# B&R Automation Studio project 8238 (part 8)

#### kgGetMachineAdressW3.st - Ermittelt die Maschinenadresse aus Liniennummer und Maschinentyp
```iecst
(********************************************************************
 * COPYRIGHT -- Herbert Kannegiesser GmbH
 ********************************************************************
 * Library: KGstdLib
 * File: kgGetMachineAdressW3.st
 * Author: hunholz
 * Created: February 08, 2012
 ********************************************************************
 * Implementation of library KGstdLib
 ********************************************************************)

(* Ermittelt die Maschinenadresse aus Liniennummer und Maschinentyp *)
FUNCTION kgGetMachineAdressW3

	_diMachineType ACCESS ADR(MachineType);

	kgGetMachineAdressW3 := 0;

	IF MachineType = kgW3SERVER THEN

		kgGetMachineAdressW3 := 202;

	ELSE

		CASE MachineType OF

			kgW3LOADSYSTEM, kgW3EXTRACTOR, kgW3EXTRACTOR2, kgW3CONVEYOR, kgW3SHAKER, kgW3PROCESS:

				IF LineNumber >= 1 AND LineNumber <= 10 THEN

					kgGetMachineAdressW3 := DINT_TO_USINT(_diMachineType) + LineNumber;

				END_IF

			kgW3WASHER, kgW3IFBOX, kgW3DEVICE, kgW3PCSTATION, kgW3BIT:

				IF LineNumber >= 1 AND LineNumber <= 20 THEN

					kgGetMachineAdressW3 := DINT_TO_USINT(_diMachineType) + LineNumber;

				END_IF

			kgW3DRYER, kgW3SINGLEWASHER:

				IF LineNumber >= 1 AND LineNumber <= 30 THEN

					kgGetMachineAdressW3 := DINT_TO_USINT(_diMachineType) + LineNumber;

				END_IF

		END_CASE

	END_IF

END_FUNCTION
```

#### kgCheckDo.st - Prüfe auf Datenobjekt und erzeuge es ggf. neu
```iecst
(********************************************************************
 * COPYRIGHT -- Herbert Kannegiesser GmbH
 ********************************************************************
 * Library: KGstdLib
 * File: kgCheckDo.st
 * Author: hunholz
 * Created: February 22, 2012
 ********************************************************************
 * Implementation of library KGstdLib
 ********************************************************************)

(* Prüfe auf Datenobjekt und erzeuge es ggf. neu *)
FUNCTION_BLOCK kgCheckDo

	IF Enable THEN

		_xReady := FALSE;

		IF MinLen > NomLen THEN

			Status := KG_ERR_WRONGSIZES;
			RETURN;

		END_IF

		REPEAT

			CASE _wStep OF

				0:	// Hole Info

					_doInfo(enable := TRUE, pName := pName);

					IF _doInfo.status = ERR_OK THEN

						IF _doInfo.len >= MinLen THEN

							doId 	:= _doInfo.ident;
							doMem 	:= _doInfo.pDatObjMem;
							doLen 	:= _doInfo.len;

							Status := ERR_OK;

							_xReady := TRUE;

						ELSE

							_wStep := 1;
							Status := ERR_OK;

						END_IF

					ELSIF _doInfo.status <> ERR_FUB_BUSY THEN

						IF Create THEN

							// DO ist nicht vorhanden

							_wStep := 2;
							Status := ERR_OK;

						ELSE

							Status := _doInfo.status;
							_xReady := TRUE;

						END_IF

					END_IF

				1:	// Lösche vorhandenes DO

					_doDelete(enable := TRUE, ident := _doInfo.ident);

					IF _doDelete.status <> ERR_FUB_BUSY THEN

						Status := ERR_OK;
						_wStep := 2;

					ELSE

						Status := ERR_FUB_BUSY;

					END_IF

				2:	// Erzeuge DO neu

					_doCreate(enable := TRUE, grp := 0, pName := pName, len := NomLen, MemType := MemType, Option := 0, pCpyData := 0);

					IF _doCreate.status = ERR_OK THEN

						_wStep := 3;

					ELSIF _doCreate.status <> ERR_FUB_BUSY THEN

						_wStep := 0;

					END_IF

					Status := _doCreate.status;

				3: // Info erneut einlesen

					_doInfo(enable := TRUE, pName := pName);

					IF _doInfo.status = ERR_OK THEN

						doId 	:= _doInfo.ident;
						doMem 	:= _doInfo.pDatObjMem;
						doLen 	:= _doInfo.len;

						Status := KG_INFO_DO_NEW;

						_xReady := TRUE;

						_wStep := 0;

					ELSIF _doInfo.status <> ERR_FUB_BUSY THEN

						Status := _doInfo.status;
						_wStep := 0;

					ELSE

						Status := _doInfo.status;

					END_IF

				ELSE

					_wStep := 0;
					Status := ERR_OK;

			END_CASE

			UNTIL

			Status <> ERR_OK OR _xReady

		END_REPEAT

	ELSE

		_wStep := 0;

		Status := ERR_FUB_ENABLE_FALSE;

	END_IF

END_FUNCTION_BLOCK
```

#### kgXOR.st - XOR über Byte-Feld
```iecst
(********************************************************************
 * COPYRIGHT -- Herbert Kannegiesser GmbH
 ********************************************************************
 * Library: KGstdLib
 * File: kgXOR.st
 * Author: hunholz
 * Created: March 07, 2012
 ********************************************************************
 * Implementation of library KGstdLib
 ********************************************************************)

(* XOR über Byte-Feld *)
FUNCTION kgXOR

	_xStatusOk := pStatus > 0;

	kgXOR := 0;

	IF _xStatusOk THEN
		_wDynStatus ACCESS pStatus;
		_wDynStatus := ERR_OK;
	END_IF

	_xWordResultOk := pWordResult > 0;

	IF _xWordResultOk THEN

		_bWordResult ACCESS pWordResult;

	END_IF

	IF pMem = 0 THEN
		IF _xStatusOk THEN
			_wDynStatus := KG_ERR_NULPOINTER;
		END_IF
		RETURN;

	ELSE

		_bMem ACCESS pMem;

	END_IF

	kgXOR := bInit;

	FOR _i := 1 TO wLen DO

		kgXOR := kgXOR XOR _bMem[_i];

	END_FOR

	IF _xWordResultOk THEN

		_bWordResult[0] := kgXOR;
		_bWordResult[1] := kgXOR;

	END_IF

END_FUNCTION
```

#### kgUnitconfREALtoDisplay.st - Wandelt Wert entsprechend der Unit
```iecst
(********************************************************************
 * COPYRIGHT -- Herbert Kannegiesser GmbH
 ********************************************************************
 * Library: KGstdLib
 * File: kgUnitconfREALtoDisplay.st
 * Author: hunholz
 * Created: March 15, 2012
 ********************************************************************
 * Implementation of library KGstdLib
 ********************************************************************)

(* Wandelt Wert entsprechend der Unit *)
FUNCTION kgUnitconfREALtoDisplay

	lDigits := 0;
	sUnit := '';

	CASE Unit OF

		2,60,70,80,91,901:

			// 1/10
			kgUnitconfREALtoDisplay := Value * 0.1;
			lDigits := 1;

			CASE Unit OF

				2:
					// Sekunden
					sUnit := 's';

				60:
					// Hertz
					sUnit := 'Hz';

				70:
					// Winkel
					sUnit := '°';

				80:
					// Prozent
					sUnit := '%';
				91:
					// Prozent
					sUnit := 'g';

			END_CASE

		90,902:
			// 1/100
			kgUnitconfREALtoDisplay := Value * 0.01;
			lDigits := 2;

			CASE Unit OF

				90:
					// g
					sUnit := 'g';

			END_CASE

		4,903:

			// 1/1000
			kgUnitconfREALtoDisplay := Value * 0.001;
			lDigits := 3;

			CASE Unit OF

				4:
					// Sekunde
					sUnit := 's';

			END_CASE

		10:
			// liter Gallonen
			IF LocUnit = KG_UNIT_US THEN
				kgUnitconfREALtoDisplay := Value * 0.2641721;
				lDigits := 1;
				sUnit := 'US gal';
			ELSE
				kgUnitconfREALtoDisplay := Value;
				sUnit := 'l';
			END_IF

		11:
			// milliliter Ounce
			IF LocUnit = KG_UNIT_US THEN
				kgUnitconfREALtoDisplay := Value * 0.03381402;
				lDigits := 3;
				sUnit := 'fl.Oz.';

			ELSE
				kgUnitconfREALtoDisplay := Value;
				sUnit := 'ml';
			END_IF

		20:
			// mm inch
			IF LocUnit = KG_UNIT_US THEN
				kgUnitconfREALtoDisplay := Value * 0.03937;
				lDigits := 2;
				sUnit := 'inch';
			ELSE
				kgUnitconfREALtoDisplay := Value;
				sUnit := 'mm';
			END_IF

		21:
			// mm cm inch
			IF LocUnit = KG_UNIT_US THEN
				kgUnitconfREALtoDisplay := Value * 0.03937;
				lDigits := 2;
				sUnit := 'inch';
			ELSE
				kgUnitconfREALtoDisplay := Value * 0.1;
				lDigits := 1;
				sUnit := 'cm';
			END_IF

		22:
			// mm dm inch
			IF LocUnit = KG_UNIT_US THEN
				kgUnitconfREALtoDisplay := Value * 0.03937;
				sUnit := 'inch';
			ELSE
				kgUnitconfREALtoDisplay := Value * 0.01;
				sUnit := 'dm';
			END_IF
			lDigits := 2;

		23:
			// mm m feet
			IF LocUnit = KG_UNIT_US THEN
				kgUnitconfREALtoDisplay := Value * 0.00328;
				sUnit := 'ft';
			ELSE
				kgUnitconfREALtoDisplay := Value * 0.001;
				sUnit := 'm';
			END_IF
			lDigits := 3;

		30:
			// 0,1kg kg lbs
			IF LocUnit = KG_UNIT_US THEN
				kgUnitconfREALtoDisplay := Value * 0.220462;
				sUnit := 'lbs';
			ELSE
				kgUnitconfREALtoDisplay := Value * 0.1;
				sUnit := 'kg';
			END_IF
			lDigits := 1;

		40:
			// 0,1 °C °C °F
			IF LocUnit = KG_UNIT_US THEN
				kgUnitconfREALtoDisplay := (Value * 0.18) + 32.0;
				sUnit := '°F';
			ELSE
				kgUnitconfREALtoDisplay := Value * 0.1;
				sUnit := '°C';
			END_IF
			lDigits := 1;

		41:
			// °C °C °F
			IF LocUnit = KG_UNIT_US THEN
				kgUnitconfREALtoDisplay := (Value * 1.8) + 32.0;
				sUnit := '°F';
			ELSE
				kgUnitconfREALtoDisplay := Value;
				sUnit := '°C';
			END_IF

		50:
			// 0,1 bar bar psi
			IF LocUnit = KG_UNIT_US THEN
				kgUnitconfREALtoDisplay := Value * 1.450368;
				sUnit := 'psi';
			ELSE
				kgUnitconfREALtoDisplay := Value * 0.1;
				lDigits := 1;
				sUnit := 'bar';
			END_IF

		310:
			// 0,01 l/kg l/kg gal/lbs
			IF LocUnit = KG_UNIT_US THEN
				kgUnitconfREALtoDisplay := Value * 0.00119827;
				lDigits := 2;
				sUnit := 'gal/lbs';
			ELSE
				kgUnitconfREALtoDisplay := Value * 0.01;
				lDigits := 1;
				sUnit := 'l/kg';
			END_IF

		ELSE

			kgUnitconfREALtoDisplay := Value;

			CASE Unit OF

				1:
					sUnit := 's';
				3:
					sUnit := 'min';
				81:
					sUnit := '%';

			END_CASE

	END_CASE

	IF pDigits > 0 THEN

		brsmemcpy(pDigits, ADR(lDigits), SIZEOF(lDigits));

	END_IF

	IF pUnit > 0 THEN

		brsmemcpy(pUnit, ADR(sUnit), SIZEOF(sUnit));

	END_IF

END_FUNCTION
```

#### kgUnitconfDisplayToREAL.st - Wandelt Wert entsprechend der Unit
```iecst
(********************************************************************
 * COPYRIGHT -- Herbert Kannegiesser GmbH
 ********************************************************************
 * Library: KGstdLib
 * File: kgUnitconfDisplayToREAL.st
 * Author: hunholz
 * Created: March 15, 2012
 ********************************************************************
 * Implementation of library KGstdLib
 ********************************************************************)

(* Wandelt Wert entsprechend der Unit *)
FUNCTION kgUnitconfDisplayToREAL

	CASE Unit OF

		2,60,70,80,91,901:
			// 1/10
			kgUnitconfDisplayToREAL := Display * 10;

		90,902:
			// 1/100
			kgUnitconfDisplayToREAL := Display * 100;

		4,903:
			// 1/1000
			kgUnitconfDisplayToREAL := Display * 1000;

		10:
			// liter Gallonen
			IF LocUnit = KG_UNIT_US THEN
				kgUnitconfDisplayToREAL := Display / 0.2641721;
			ELSE
				kgUnitconfDisplayToREAL := Display;
			END_IF

		11:
			// milliliter Ounce
			IF LocUnit = KG_UNIT_US THEN
				kgUnitconfDisplayToREAL := Display / 0.03381402;
			ELSE
				kgUnitconfDisplayToREAL := Display;
			END_IF

		20:
			// mm inch
			IF LocUnit = KG_UNIT_US THEN
				kgUnitconfDisplayToREAL := Display / 0.03937;
			ELSE
				kgUnitconfDisplayToREAL := Display;
			END_IF

		21:
			// mm cm inch
			IF LocUnit = KG_UNIT_US THEN
				kgUnitconfDisplayToREAL := Display / 0.03937;
			ELSE
				kgUnitconfDisplayToREAL := Display * 10;
			END_IF

		22:
			// mm dm inch
			IF LocUnit = KG_UNIT_US THEN
				kgUnitconfDisplayToREAL := Display / 0.03937;
			ELSE
				kgUnitconfDisplayToREAL := Display * 100;
			END_IF

		23:
			// mm m feet
			IF LocUnit = KG_UNIT_US THEN
				kgUnitconfDisplayToREAL := Display / 0.00328;
			ELSE
				kgUnitconfDisplayToREAL := Display * 1000;
			END_IF

		30:
			// 0,1kg kg lbs
			IF LocUnit = KG_UNIT_US THEN
				kgUnitconfDisplayToREAL := Display / 0.220462;
			ELSE
				kgUnitconfDisplayToREAL := Display * 10;
			END_IF

		40:
			// 0,1 °C °C °F
			IF LocUnit = KG_UNIT_US THEN
				kgUnitconfDisplayToREAL := (Display - 32.0) / 0.18;
			ELSE
				kgUnitconfDisplayToREAL := Display * 10;
			END_IF

		41:
			// °C °C °F
			IF LocUnit = KG_UNIT_US THEN
				kgUnitconfDisplayToREAL := (Display - 32.0) / 1.8;
			ELSE
				kgUnitconfDisplayToREAL := Display;
			END_IF

		50:
			// 0,1 bar bar psi
			IF LocUnit = KG_UNIT_US THEN
				kgUnitconfDisplayToREAL := Display / 1.450368;
			ELSE
				kgUnitconfDisplayToREAL := Display * 10;
			END_IF

		310:
			// 0,01 l/kg l/kg gal/lbs
			IF LocUnit = KG_UNIT_US THEN
				kgUnitconfDisplayToREAL := Display / 0.00119827;
			ELSE
				kgUnitconfDisplayToREAL := Display * 100;
			END_IF

		ELSE

			kgUnitconfDisplayToREAL := Display;

	END_CASE

END_FUNCTION
```

#### kgGetProgdata.st - Read Programdata from a dataobject
```iecst
(********************************************************************
 * COPYRIGHT -- Herbert Kannegiesser GmbH
 ********************************************************************
 * Library: KGstdLib
 * File: kgGetProgdata.st
 * Author: hunholz
 * Created: April 11, 2012
 ********************************************************************
 * Implementation of library KGstdLib
 ********************************************************************)

(* Read Programdata from a dataobject *)
FUNCTION kgGetProgdata

	IF LEN(sBaseName) = 0 THEN
		kgGetProgdata := KG_ERR_NULLSTRING;
		RETURN;
	END_IF

	IF pMem = 0 THEN
		kgGetProgdata := KG_ERR_NULPOINTER;
		RETURN;
	END_IF

	_sIndex := '';
	IF wProgMaxNo > 9999 AND  wProgNo  < 10000 THEN
		_sIndex := CONCAT(_sIndex,'0');
	END_IF
	IF wProgMaxNo > 999 AND  wProgNo  < 1000 THEN
		_sIndex := CONCAT(_sIndex,'0');
	END_IF
	IF wProgMaxNo > 99 AND  wProgNo  < 100 THEN
		_sIndex := CONCAT(_sIndex,'0');
	END_IF
	IF wProgMaxNo > 9 AND  wProgNo  < 10 THEN
		_sIndex := CONCAT(_sIndex,'0');
	END_IF

	_sIndex1 := UINT_TO_STRING(wProgNo);

	_sIndex := CONCAT(_sIndex, _sIndex1);

	_sName := CONCAT(sBaseName, _sIndex);

	_diProg(enable := TRUE, pName := ADR(_sName));

	IF _diProg.status = ERR_OK THEN

		// Bug 690 : Datenobjekt hat 4Byte Alignment. Struktur kann 1 bis 3 Byte kleiner sein.
//		IF _diProg.len > lSize THEN
//			kgGetProgdata := KG_ERR_WRONGSIZES;
//			RETURN;
//		END_IF

		brsmemcpy(pMem, _diProg.pDatObjMem, MIN(_diProg.len,lSize));

		kgGetProgdata := ERR_OK;

		RETURN;

	ELSE
		kgGetProgdata := _diProg.status;
		RETURN;
	END_IF

END_FUNCTION
```

#### kgSignalLight.st - Process red/yellow/green
```iecst
(********************************************************************
 * COPYRIGHT -- Herbert Kannegiesser GmbH
 ********************************************************************
 * Library: KGstdLib
 * File: kgSignalLight.st
 * Author: hunholz
 * Created: July 12, 2012
 ********************************************************************
 * Implementation of library KGstdLib
 ********************************************************************)

(* Process red/yellow/green *)
FUNCTION kgSignalLight

	xGreen 		:= FALSE;
	xRed		:= FALSE;
	xYellow 	:= FALSE;

	CASE wStatus OF

		(*-0- Maschine aus*)
		KG_MACHINESTATE_OFF:

		(*-1- NOT-HALT*)
		KG_MACHINESTATE_EMERGENCYSTOP:

			xRed := xClock;

		(*-2- Sicherer HALT*)
		KG_MACHINESTATE_SAFESTOP:

			xYellow := xClock;

		(*-3- Störung*)
		KG_MACHINESTATE_FAULT:

			xRed := TRUE;

		(*-4- Störung quittierbar*)
		KG_MACHINESTATE_FAULT_GONE:

			xRed := TRUE;
			xYellow := xClock;

		(*-5- Service / Handbetrieb*)
		KG_MACHINESTATE_SERVICE:

			xYellow := xClock;
			xGreen := xClock;

		(*-6- Maschine läuft*)
		KG_MACHINESTATE_AUTOMATIC_RUN:

			xGreen := TRUE;

		(*-7- STOP*)
		KG_MACHINESTATE_STOP:

		(*-8- Maschine wartet auf Automatik-Freigabe*)
		KG_MACHINESTATE_WAIT_AUTOMATIC:

			xGreen := xClock;

		(*-9- Maschine wartet auf Bestätigung durch Bediener*)
		KG_MACHINESTATE_WAIT_MAN:

			xYellow := xClock;
			xGreen := TRUE;

		(*-10- Warnung*)
		KG_MACHINESTATE_WARNING:

			xYellow := TRUE;
			xGreen := TRUE;

		ELSE

			xGreen := TRUE;

	END_CASE

END_FUNCTION
```

### KGStandard-History.txt
```
1.00.0	30.06.2011 NEU
1.01.0	02.07.2011 mnCnt ergänzt
1.02.0	08.07.2011 Netlink 1.02.0
1.03.0  19.07.2011 kgStd 1.01.0
1.04.0	26.07.2011 Maschinentyp in der Infostruktur auf 11 Zeichen verringert
1.05.0		   Keine Ahnung
1.06.0	01.09.2011 Info_typ erweitert
1.07.0	20.09.2011 Stat_typ ergänzt
1.08.0	06.10.2011 Netlink 1.05.0
1.08.1	14.10.2011 Netlink 1.06.0
1.09.0  03.11.2011 Umstellung auf AS 3.0.90
					- Stat_typ erweitert
					- Funktionen zum Generieren einer Postennummer in KGstdLib ergänzt 1.02.0
1.10.0	20.12.2011 Ringbufferfunktionen ergänzt
				   KGBOM ergänzt
				   KG_DEVICE_COMPACTFLASH ergänzt
1.11.0	03.01.2012 kgGUIDisZero : Funktion prüft, ob eine GUID null ist.
1.12.0	12.01.2012 kgNextBatchNoLong merkt sich die letzte Postennummer. BatchNo ist nur noch Output.
1.13.0	24.01.2012 Erweiterung der Ringbuffer-Funktionen. Einführung des Startzeigers.
				   Unabhängigkeit von Netlink. Netlink entfernt.
				   Konstanten für Maschinenstati ergänzt
				   Maschinentypen aus NetLink-Library übernommen. nlMachinetypeW3_typ --> kgMachinetypeW3_typ
				   Datentypen utfName15 und utfName31 als abgeleiteten Datentyp deklariert
1.14.0	03.02.2012 Im Pkg_KGStandardShare werden die Konstanten KG_DEVICE_USBSTICK1 und KG_DEVICE_USBSTICK2 als STRING[31] deklariert.
				   In der sysconf sollten die Device-Namen für gültige USB-Massenspeicher definiert sein.
1.15.0	08.02.2012 Funktionen: kgGetLineNumberW3 und kgGetMachineAdressW3. (mnEth Version 2.08.0 verwenden)
1.15.1	15.02.2012 kgGetBatchNoUnique und kgNextBatchNoLong korrigiert
1.16.0	15.03.2012 Konvertierung von Parametern entsprechend der Einheit (units.csv 2011-11-25T08:56:00)
1.16.1	15.03.2012 Für Displaywerte werden auch die Nachkommastellen mit angegeben
1.16.2	20.03.2012 Bugfix KGstdLib
1.17.0	21.03.2012 KGstdLib erweitert
1.17.1	22.03.2012 CP3585 ergänzt
1.18.0	04.04.2012 _Info_ gibt es nicht mehr
1.19.0	11.04.2012 Enumeration für Maschinenstati
1.20.0	04.05.2012 Einheit (91) 0,1 g ergänzt
1.21.0	18.06.2012 CP1584 ergänzt
		19.06.2012 Bug 690: Programm lässt sich nicht laden behoben
		21.06.2012 Maschinenstati in Hex-Notation und als USINT. Erweiterter Maschinenstatus als UINT mit Bit 8 für Stop und Bit 9 für Warten
1.22.0	25.06.2012 Module Identifier ergänzt (X20DI9371, X20DO9322)
1.23.0	03.07.2012 Module Identifier ergänzt (X20IF1072, X20IF2772, X20BR9300, X20PS2100, 4PP065IF231
1.24.0	18.07.2012 Module Identifier ergänzt (X20BT9400, X67DM1321
1.25.0	18.09.2012 CP3484 ergänzt
```

### Package Logical/Standard/Kanlink/KGFramework/Pkg_mnSystem - Systemtask für Versionierung

### Program Logical/Standard/Kanlink/KGFramework/Pkg_mnSystem/mnSystem (IEC) - Systemtask für Versionierung

#### mnSystemCyclic.st - Cyclic code
```iecst
(********************************************************************
 * COPYRIGHT -- Kannegiesser GmbH
 ********************************************************************
 * Program: mnSystem
 * File: mnSystemCyclic.st
 * Author: Hunholz
 * Created: Mar 16, 2012
 ********************************************************************
 * Implementation of program mnSystem
 ********************************************************************)

PROGRAM _CYCLIC

	//**********************
	// USB Knoten überwachen
	//**********************

	// Alle 5 Sekunden eine Liste der verfügbaren Sticks zur Verfügung stellen

	_TONsearchForUSB(IN := _wUSBstate = 0 , PT := T#5s);

	CASE _wUSBstate OF

		0:

			IFmnSystem.Out.sInterfaceUSB := _sInterfaceUSB;
			IFmnSystem.Out.xUSBStickReady := _xUSBStickReady;

			IF _TONsearchForUSB.Q OR _xFirstScan THEN

				_xFirstScan := FALSE;
				_wUSBstate := 1;

			END_IF

		1:
			_UsbNodeListGet(enable := TRUE, pBuffer := ADR(_lUSBlist), bufferSize := SIZEOF(_lUSBlist), filterInterfaceClass := asusb_CLASS_MASS_STORAGE, filterInterfaceSubClass := asusb_SUBCLASS_SCSI_COMMAND_SET);

			IF _UsbNodeListGet.status <> ERR_FUB_BUSY THEN

				_sInterfaceUSB := '';
				_xUSBStickReady := FALSE;

				IF _UsbNodeListGet.status = ERR_OK THEN

					_wUSBstate := 2;

					_wCycleFound := _wCycleFound + 1;

				ELSE

					IFmnSystem.Out.xUSBStickScanned := TRUE;
					_wUSBstate := 0;

					_wCycleNotFound := _wCycleNotFound + 1;

				END_IF

			END_IF

		2:

			_UsbNodeGet(enable := TRUE, nodeId := _lUSBlist[1], pBuffer := ADR(_usbNode), bufferSize := SIZEOF(_usbNode));

			IF _UsbNodeGet.status <> ERR_FUB_BUSY THEN

				IF _UsbNodeGet.status = ERR_OK THEN

					brsmemcpy(ADR(_sInterfaceUSB),ADR(_usbNode.ifName),SIZEOF(_sInterfaceUSB));
					_xUSBStickReady := TRUE;

					_wCycleReady := _wCycleReady + 1;

				END_IF

				IFmnSystem.Out.xUSBStickScanned := TRUE;
				IFmnSystem.Out.sInterfaceUSB := _sInterfaceUSB;
				IFmnSystem.Out.xUSBStickReady := _xUSBStickReady;

				_wUSBstate := 0;

			END_IF

		ELSE

			_wUSBstate := 0;

	END_CASE

	//#####################################################################################################################

	// Heartbeeat erzeugen (Sekunden)
	_GetTime(enable := TRUE);
	mnSystemStatAd.wHeartbeat := DT_TO_UINT(_GetTime.DT1);

	_diDifSystime := IFmnSystem.In.PLC.diSystemTime - _diOldSysTime;
	_diOldSysTime := IFmnSystem.In.PLC.diSystemTime;

	IF _diDifSystime >= 0 THEN

		_l1sCount := _l1sCount + DINT_TO_UDINT(_diDifSystime);

		IF _l1sCount > 1000000 THEN

			IFmnSystem.Out.x1s := NOT IFmnSystem.Out.x1s;
			_l1sCount := _l1sCount - 1000000;

		END_IF

		_l500msCount := _l500msCount + DINT_TO_UDINT(_diDifSystime);

		IF _l500msCount > 500000 THEN

			IFmnSystem.Out.x500ms := NOT IFmnSystem.Out.x500ms;
			_l500msCount := _l500msCount - 500000;

		END_IF

	END_IF

	// Lüfterüberwachung

	CASE IFmnSystem.In.PLC.wMDL_ID OF

		KG_CPU_X20CP1486:

			_xFanOk := IFmnSystem.In.PLC.xFanOk;

		ELSE

			_xFanOk := TRUE;

	END_CASE

	//********************************
	// Überwachung Umgebungstemperatur
	//********************************

	_TONtemp(IN := (IFmnSystem.In.PLC.wTemperatureENV > mnSystemPar.Mac.wWarnTemperatureEnvironment) AND IFmnParam.Out.xParamOK, PT := T#10m);
	_TONtempC(IN := (IFmnSystem.In.PLC.wTemperatureENV > (mnSystemPar.Mac.wWarnTemperatureEnvironment - 50)) AND IFmnParam.Out.xParamOK, PT := T#10m);

	//************************
	// Überwachung von Modulen
	//************************

	IF IFmnParam.Out.xParamOK THEN

		_xModuleFault := FALSE;
		_wModuleFaultLineNumber := 0;
		_wModuleFaultModuleNumber := 0;

		FOR _ii := 1 TO MNSYSTEM_CNT_MODULELINES DO

			FOR _jj := 1 TO MNSYSTEM_CNT_MODULES DO

				IF mnSystemPar.Cfg.Lines[_ii].wModuleID[_jj] <> KG_MODULE_NO THEN

					// Modul ist konfiguriert

					IF (mnSystemPar.Cfg.Lines[_ii].wModuleID[_jj] <> IFmnSystem.In.ModuleInfo[_ii,_jj].wMDL_ID) THEN
						_xModuleFault := TRUE;
						_wModuleFaultLineNumber := _ii;
						_wModuleFaultModuleNumber := _jj;
						EXIT;
					END_IF

				END_IF

			END_FOR

			IF _xModuleFault THEN
				EXIT;
			END_IF

		END_FOR

		// Cooling

		FOR _iC := 1 TO 2 DO

			IF NOT _xCInitDone[_iC] THEN

				IF mnSystemPar.Cfg.BindingMotProtCooling[_iC].wBindIndexModul > 0 AND mnSystemPar.Cfg.BindingMotProtCooling[_iC].wBindIndexModul <= MNSYSTEM_CNT_MODULES
					AND mnSystemPar.Cfg.BindingMotProtCooling[_iC].wBindIndexChannel > 0 AND mnSystemPar.Cfg.BindingMotProtCooling[_iC].wBindIndexChannel <= 12 THEN

					_BindMotProtCooling[_iC].wModule := mnSystemPar.Cfg.BindingMotProtCooling[_iC].wBindIndexModul;
					_BindMotProtCooling[_iC].wChannel := mnSystemPar.Cfg.BindingMotProtCooling[_iC].wBindIndexChannel;
					_BindMotProtCooling[_iC].sDiscription := mnSystemPar.Cfg.BindingMotProtCooling[_iC].sDiscription;
					_BindMotProtCooling[_iC].xInvers := mnSystemPar.Cfg.BindingMotProtCooling[_iC].xInvers;
					_BindMotProtCooling[_iC].xQualitiyOk := TRUE;

				END_IF

				IF mnSystemPar.Cfg.BindingOutCooling[_iC].wBindIndexModul > 0 AND mnSystemPar.Cfg.BindingOutCooling[_iC].wBindIndexModul <= MNSYSTEM_CNT_MODULES
					AND mnSystemPar.Cfg.BindingOutCooling[_iC].wBindIndexChannel > 0 AND mnSystemPar.Cfg.BindingOutCooling[_iC].wBindIndexChannel <= 12 THEN

					_BindingOutCooling[_iC].wModule := mnSystemPar.Cfg.BindingOutCooling[_iC].wBindIndexModul;
					_BindingOutCooling[_iC].wChannel := mnSystemPar.Cfg.BindingOutCooling[_iC].wBindIndexChannel;
					_BindingOutCooling[_iC].sDiscription := mnSystemPar.Cfg.BindingOutCooling[_iC].sDiscription;
					_BindingOutCooling[_iC].xInvers := mnSystemPar.Cfg.BindingOutCooling[_iC].xInvers;
					_BindingOutCooling[_iC].xQualitiyOk := TRUE;

				END_IF

				IF mnSystemPar.Cfg.BindingWarnEnvTemp[_iC].wBindIndexModul > 0 AND mnSystemPar.Cfg.BindingWarnEnvTemp[_iC].wBindIndexModul <= MNSYSTEM_CNT_MODULES
					AND mnSystemPar.Cfg.BindingWarnEnvTemp[_iC].wBindIndexChannel > 0 AND mnSystemPar.Cfg.BindingWarnEnvTemp[_iC].wBindIndexChannel <= 12 THEN

					_BindingWarnEnvTemp[_iC].wModule := mnSystemPar.Cfg.BindingWarnEnvTemp[_iC].wBindIndexModul;
					_BindingWarnEnvTemp[_iC].wChannel := mnSystemPar.Cfg.BindingWarnEnvTemp[_iC].wBindIndexChannel;
					_BindingWarnEnvTemp[_iC].sDiscription := mnSystemPar.Cfg.BindingWarnEnvTemp[_iC].sDiscription;
					_BindingWarnEnvTemp[_iC].xInvers := mnSystemPar.Cfg.BindingWarnEnvTemp[_iC].xInvers;
					_BindingWarnEnvTemp[_iC].xQualitiyOk := TRUE;

				END_IF

				_xCInitDone[_iC] := TRUE;

			ELSE

				IF _BindMotProtCooling[_iC].xQualitiyOk THEN

					_xFaultMotProtCooling[_iC] := MDLIn[1,_BindMotProtCooling[_iC].wModule].xIn[_BindMotProtCooling[_iC].wChannel] XOR _BindMotProtCooling[_iC].xInvers;

				ELSE

					_xFaultMotProtCooling[_iC] := FALSE;

				END_IF

				IF _BindingWarnEnvTemp[_iC].xQualitiyOk THEN

					_xWarnEnvTemp[_iC] := MDLIn[1,_BindingWarnEnvTemp[_iC].wModule].xIn[_BindingWarnEnvTemp[_iC].wChannel] XOR _BindingWarnEnvTemp[_iC].xInvers;

				ELSE

					_xWarnEnvTemp[_iC] := FALSE;

				END_IF

				IF _BindingOutCooling[_iC].xQualitiyOk THEN

					MDLOut[1,_BindingOutCooling[_iC].wModule].xOut[_BindingOutCooling[_iC].wChannel] := (NOT _xFaultMotProtCooling[_iC] AND (_xWarnEnvTemp[_iC] OR (_TONtempC.Q AND (_iC = 1))))
																											XOR _BindingOutCooling[_iC].xInvers;

				END_IF

			END_IF

		END_FOR

	ELSE

		_xModuleFault := FALSE;
		_wModuleFaultLineNumber := 0;
		_wModuleFaultModuleNumber := 0;

	END_IF

	// Meldungen
	IF NOT IFmnTest.Out.xNoMessages THEN

		kgMsgStatus[MNSYSTEM_IDX_KGMSGSTAT].wFunction_ID 	:= 110;

		IF _xModuleFault THEN

			kgMsgStatus[MNSYSTEM_IDX_KGMSGSTAT].wMsgClass		:= MNMSG_CLASS_WARNING;
			kgMsgStatus[MNSYSTEM_IDX_KGMSGSTAT].wMsgAckLevel	:= 0;
			kgMsgStatus[MNSYSTEM_IDX_KGMSGSTAT].wMsgNumber		:= MNSYSTEM_MSG_WRONGMODULE;
			kgMsgStatus[MNSYSTEM_IDX_KGMSGSTAT].diMsgAttr1		:= _wModuleFaultLineNumber;
			kgMsgStatus[MNSYSTEM_IDX_KGMSGSTAT].diMsgAttr2		:= _wModuleFaultModuleNumber;
			kgMsgStatus[MNSYSTEM_IDX_KGMSGSTAT].sMsgAttrTxt		:= mnSystemPar.Cfg.Lines[_wModuleFaultLineNumber].sName[_wModuleFaultModuleNumber];

		ELSIF NOT _xFanOk THEN

			kgMsgStatus[MNSYSTEM_IDX_KGMSGSTAT].wMsgClass		:= MNMSG_CLASS_WARNING;
			kgMsgStatus[MNSYSTEM_IDX_KGMSGSTAT].wMsgAckLevel	:= 0;
			kgMsgStatus[MNSYSTEM_IDX_KGMSGSTAT].wMsgNumber		:= MNSYSTEM_MSG_FAN;
			kgMsgStatus[MNSYSTEM_IDX_KGMSGSTAT].diMsgAttr1		:= 0;
			kgMsgStatus[MNSYSTEM_IDX_KGMSGSTAT].diMsgAttr2		:= 0;
			kgMsgStatus[MNSYSTEM_IDX_KGMSGSTAT].sMsgAttrTxt		:= '';

		ELSIF _xFaultMotProtCooling[1] OR _xFaultMotProtCooling[1] THEN

			kgMsgStatus[MNSYSTEM_IDX_KGMSGSTAT].wMsgClass		:= MNMSG_CLASS_WARNING;
			kgMsgStatus[MNSYSTEM_IDX_KGMSGSTAT].wMsgAckLevel	:= 0;
			kgMsgStatus[MNSYSTEM_IDX_KGMSGSTAT].wMsgNumber		:= MNSYSTEM_MSG_MOTPROTCOOLING;
			kgMsgStatus[MNSYSTEM_IDX_KGMSGSTAT].diMsgAttr1		:= 0;
			kgMsgStatus[MNSYSTEM_IDX_KGMSGSTAT].diMsgAttr2		:= 0;
			IF _xFaultMotProtCooling[1] THEN
				kgMsgStatus[MNSYSTEM_IDX_KGMSGSTAT].sMsgAttrTxt		:= _BindMotProtCooling[1].sDiscription;
			ELSE
				kgMsgStatus[MNSYSTEM_IDX_KGMSGSTAT].sMsgAttrTxt		:= _BindMotProtCooling[2].sDiscription;
			END_IF

		ELSIF _TONtemp.Q OR _xWarnEnvTemp[1] OR _xWarnEnvTemp[2] THEN

			kgMsgStatus[MNSYSTEM_IDX_KGMSGSTAT].wMsgClass		:= MNMSG_CLASS_WARNING;
			kgMsgStatus[MNSYSTEM_IDX_KGMSGSTAT].wMsgAckLevel	:= 0;
			kgMsgStatus[MNSYSTEM_IDX_KGMSGSTAT].wMsgNumber		:= MNSYSTEM_MSG_ENVTEMP;
			kgMsgStatus[MNSYSTEM_IDX_KGMSGSTAT].diMsgAttr1		:= 0;
			kgMsgStatus[MNSYSTEM_IDX_KGMSGSTAT].diMsgAttr2		:= 0;
			IF _xWarnEnvTemp[1] THEN
				kgMsgStatus[MNSYSTEM_IDX_KGMSGSTAT].sMsgAttrTxt		:= mnSystemPar.Cfg.sSwitchBoxName[1];
			ELSIF _xWarnEnvTemp[2] THEN
				kgMsgStatus[MNSYSTEM_IDX_KGMSGSTAT].sMsgAttrTxt		:= mnSystemPar.Cfg.sSwitchBoxName[2];
			ELSE
				kgMsgStatus[MNSYSTEM_IDX_KGMSGSTAT].sMsgAttrTxt		:= 'CPU';
			END_IF

		ELSIF IFmnSystem.In.PLC.bBatteryStatusCPU <> 1 THEN

			kgMsgStatus[MNSYSTEM_IDX_KGMSGSTAT].wMsgClass		:= MNMSG_CLASS_WARNING;
			kgMsgStatus[MNSYSTEM_IDX_KGMSGSTAT].wMsgAckLevel	:= 0;
			kgMsgStatus[MNSYSTEM_IDX_KGMSGSTAT].wMsgNumber		:= MNSYSTEM_MSG_BATTERY;
			kgMsgStatus[MNSYSTEM_IDX_KGMSGSTAT].diMsgAttr1		:= 0;
			kgMsgStatus[MNSYSTEM_IDX_KGMSGSTAT].diMsgAttr2		:= 0;
			kgMsgStatus[MNSYSTEM_IDX_KGMSGSTAT].sMsgAttrTxt		:= '';

		ELSE

			kgMsgStatus[MNSYSTEM_IDX_KGMSGSTAT].wFunction_ID 	:= 110;
			kgMsgStatus[MNSYSTEM_IDX_KGMSGSTAT].wMsgClass		:= 0;
			kgMsgStatus[MNSYSTEM_IDX_KGMSGSTAT].wMsgAckLevel	:= 0;
			kgMsgStatus[MNSYSTEM_IDX_KGMSGSTAT].wMsgNumber		:= 0;
			kgMsgStatus[MNSYSTEM_IDX_KGMSGSTAT].diMsgAttr1		:= 0;
			kgMsgStatus[MNSYSTEM_IDX_KGMSGSTAT].diMsgAttr2		:= 0;
			kgMsgStatus[MNSYSTEM_IDX_KGMSGSTAT].sMsgAttrTxt		:= '';

		END_IF

	END_IF

	// Stati
	mnSystemStatAd.lSerialNumber 			:= IFmnSystem.In.PLC.lSerialNumber;
	mnSystemStatAd.wTemperatureCPU 			:= IFmnSystem.In.PLC.wTemperatureCPU;
	mnSystemStatAd.wTemperatureEnvironment 	:= IFmnSystem.In.PLC.wTemperatureENV;

	// Interface
	IFmnSystem.Out.xModuleFault				:= _xModuleFault;

END_PROGRAM
```

#### mnSystemInit.st - Initialization code
```iecst
(********************************************************************
 * COPYRIGHT -- Kannegiesser GmbH
 ********************************************************************
 * Program: mnSystem
 * File: mnSystemInit.st
 * Author: horn
 * Created: January 10, 2012
 ********************************************************************
 * Implementation of program mnSystem
 ********************************************************************)

PROGRAM _INIT

	// Packet-Version auslesen mit MO_ver aus SYS_lib und für den Additional Status zur Verfügung stellen

	_sPkgName := 'mnSystem';

	IF ( MO_ver(ADR(_sPkgName), 0, ADR(_VerStruc)) = 0 ) THEN

		brsmemcpy(ADR(mnSystemStatAd.sPkgVersion), ADR(_VerStruc.version), SIZEOF(_VerStruc.version));

	ELSE

		mnSystemStatAd.sPkgVersion := '---';

	END_IF

	_sPkgName := 'mnMaster';

	IF ( MO_ver(ADR(_sPkgName), 0, ADR(_VerStruc)) = 0 ) THEN

		brsmemcpy(ADR(mnSystemStatAd.sPrjVersion), ADR(_VerStruc.version), SIZEOF(_VerStruc.version));

	ELSE

		mnSystemStatAd.sPrjVersion := '---';

	END_IF

	_sPkgName := 'mnTest';

	IF ( MO_ver(ADR(_sPkgName), 0, ADR(_VerStruc)) = 0 ) THEN

		brsmemcpy(ADR(mnSystemStatAd.sFWVersion), ADR(_VerStruc.version), SIZEOF(_VerStruc.version));

	ELSE

		mnSystemStatAd.sFWVersion := '---';

	END_IF

	// CPU-Typ bestimmen

	CASE IFmnSystem.In.PLC.wMDL_ID OF

		KG_CPU_CTT_11:

			mnSystemStatAd.sCPUType := 'CTT-11';

		KG_CPU_PCT_03:

			mnSystemStatAd.sCPUType := 'PCT-03';

		KG_CPU_PCT_04:

			mnSystemStatAd.sCPUType := 'PCT-04';

		KG_CPU_PP65_0571_P74:

			mnSystemStatAd.sCPUType := 'PP65.0571.P74';

		KG_CPU_PP420_1043_75:

			mnSystemStatAd.sCPUType := 'PP420.1043.75';

		KG_CPU_X20CP1484:

			mnSystemStatAd.sCPUType := 'CP1484';

		KG_CPU_X20CP1484_1:

			mnSystemStatAd.sCPUType := 'CP1484-1';

		KG_CPU_X20CP1486:

			mnSystemStatAd.sCPUType := 'CP1486';

		KG_CPU_X20CP3484:

			mnSystemStatAd.sCPUType := 'CP3484';

		KG_CPU_X20CP3484_1:

			mnSystemStatAd.sCPUType := 'CP3484-1';

		KG_CPU_X20CP3486:

			mnSystemStatAd.sCPUType := 'CP3486';

		KG_CPU_X20CP3585:

			mnSystemStatAd.sCPUType := 'CP3585';

		KG_CPU_X20CP1584:

			mnSystemStatAd.sCPUType := 'CP1584';

		ELSE

			mnSystemStatAd.sCPUType := UINT_TO_STRING(IFmnSystem.In.PLC.wMDL_ID);

	END_CASE

	_wMdlId := IFmnSystem.In.PLC.wMDL_ID;

END_PROGRAM
```

#### mnSystem.typ - Local data types
```iecst
(********************************************************************
 * COPYRIGHT -- Kannegiesser GmbH
 ********************************************************************
 * Program: mnSystem
 * File: _mnSystem.typ
 * Author: horn
 * Created: January 10, 2012
 ********************************************************************
 * Local data types of program mnSystem
 ********************************************************************)

TYPE
	_mnSystemMdlBind_typ : 	STRUCT
		wModule : UINT;
		wChannel : UINT;
		sDiscription : STRING[13];
		xInvers : BOOL;
		xQualitiyOk : BOOL;
	END_STRUCT;
END_TYPE
```

#### mnSystem.var - Local variables
```iecst
(********************************************************************
 * COPYRIGHT -- Kannegiesser GmbH
 ********************************************************************
 * Program: mnSystem
 * File: _mnSystem.var
 * Author: horn
 * Created: January 10, 2012
 ********************************************************************
 * Local variables of program mnSystem
 ********************************************************************)
VAR
	_sPkgName : STRING[11];
	_VerStruc : MoVerStruc_typ;
	_GetTime : DTGetTime;
	_xFanOk : BOOL;
	_wMdlId : UINT;
	_TONtemp : TON;
	_wUSBstate : UINT;
	_TONsearchForUSB : TON;
	_lUSBlist : ARRAY[1..3] OF UDINT;
	_UsbNodeListGet : UsbNodeListGet;
	_sInterfaceUSB : STRING[31];
	_xUSBStickReady : BOOL;
	_usbNode : usbNode_typ;
	_UsbNodeGet : UsbNodeGet;
	_xFirstScan : BOOL := TRUE;
	_wCycleFound : UINT;
	_wCycleNotFound : UINT;
	_wCycleReady : UINT;
	_xModuleFault : BOOL;
	_wModuleFaultLineNumber : UINT;
	_wModuleFaultModuleNumber : UINT;
	_ii : UINT;
	_jj : UINT;
	_iC : UINT;
	_xCInitDone : ARRAY[1..2] OF BOOL;
	_BindMotProtCooling : ARRAY[1..2] OF _mnSystemMdlBind_typ;
	_BindingOutCooling : ARRAY[1..2] OF _mnSystemMdlBind_typ;
	_BindingWarnEnvTemp : ARRAY[1..2] OF _mnSystemMdlBind_typ;
	_xFaultMotProtCooling : ARRAY[1..2] OF BOOL;
	_xWarnEnvTemp : ARRAY[1..2] OF BOOL;
	_TONtempC : TON;
	_diDifSystime : DINT;
	_diOldSysTime : DINT;
	_l1sCount : UDINT;
	_l500msCount : UDINT;
END_VAR
```

### Pkg_mnSystem.typ - Local data types
```iecst
(********************************************************************
 * COPYRIGHT -- Kannegiesser GmbH
 ********************************************************************
 * Program: mnSystem
 * File: mnSystem.typ
 * Author: horn
 * Created: January 10, 2012
 ********************************************************************
 * Local data types of program mnSystem
 ********************************************************************)

TYPE
	mnSystemStatAd_typ : 	STRUCT
		sPkgVersion : STRING[10]; (*Version des Packes mnSystem*)
		sPrjVersion : STRING[10]; (*Hauptversion des Projektes*)
		sFWVersion : STRING[10]; (*Frameworkversion abgeleitet aus mnTest*)
		sCPUType : STRING[19]; (*CPU-Typ*)
		wHeartbeat : UINT; (*Zählt sekündlich hoch*)
		wTemperatureCPU : UINT; (*CPU Temperatur 1/10 °C*)
		wTemperatureEnvironment : UINT; (*Umgebungstemperatur 1/10 °C*)
		lSerialNumber : UDINT; (*Seriennummer der CPU*)
	END_STRUCT;
	IFmnSystem_typ : 	STRUCT
		In : IFmnSystemIn_typ;
		Out : IFmnSystemOut_typ;
	END_STRUCT;
	IFmnSystemOut_typ : 	STRUCT
		xUSBStickReady : BOOL; (*USB-Stick erkannt*)
		xUSBStickScanned : BOOL; (*USB-Stick-Scan wurde erstmals durchgeführt*)
		xModuleFault : BOOL;
		sInterfaceUSB : STRING[31]; (*Interfacebezeichnung für den Stick*)
		x1s : BOOL;
		x500ms : BOOL;
	END_STRUCT;
	IFmnSystemIn_typ : 	STRUCT
		PLC : mnSystem_PLC_typ;
		ModuleInfo : ARRAY[1..MNSYSTEM_CNT_MODULELINES,1..MNSYSTEM_CNT_MODULES]OF mnSystem_ModuleInfo_typ;
		ModuleStatus : ARRAY[1..MNSYSTEM_CNT_MODULELINES,1..MNSYSTEM_CNT_MODULES]OF mnSystem_ModuleStatus_typ;
		xSupplyFault : ARRAY[1..12]OF BOOL;
	END_STRUCT;
	mnSystem_PLC_typ : 	STRUCT
		lSerialNumber : UDINT; (*Serien-Nummer des X20 Moduls*)
		wMDL_ID : UINT; (*Modul-ID des X20 Moduls*)
		bModeSwitch : USINT; (*Version der Firmware*)
		bBatteryStatusCPU : USINT; (*Status der Pufferbatterie*)
		xFanOk : BOOL; (*Status des CPU-Lüfters*)
		wTemperatureCPU : UINT; (*CPU-Temperatur*)
		wTemperatureENV : UINT;
		diSystemTime : DINT; (*Systemzeit der CPU in µs*)
		xStatusInput01 : BOOL; (*Status der 24V-Versorgung für I/O*)
		lPowerOnCycles : UDINT;
		lOperatingHoursPP : UDINT;
	END_STRUCT;
	mnSystem_ModuleStatus_typ : 	STRUCT
		xiMDL_OK : BOOL; (*Status des Moduls*)
		xiStatIn01 : BOOL; (*Busversorgungswarnung (1 = Ueberstrom >2,3 A oder Unterspannung <4,7 V) *)
		xiStatIn02 : BOOL; (*I/O Versorgungswarnung (0 = DC OK)*)
		aiStatus : USINT; (*Status bei Temperatur Modul*)
		xiSingleStatus : ARRAY[1..12]OF BOOL; (*Status bei digitalen Ausgängen*)
	END_STRUCT;
	mnSystem_ModuleInfo_typ : 	STRUCT
		lSerialNumber : UDINT; (*Serien-Nummer des X20 Moduls*)
		wMDL_ID : UINT; (*Modul-ID des X20 Moduls*)
		wHwVariant : UINT; (*Hardware Variante des X20 Moduls*)
		wFirmwareVers : UINT; (*Version der Firmware*)
	END_STRUCT;
	mnSystem_SignalIn_typ : 	STRUCT
		xIn : ARRAY[1..12]OF BOOL;
		iIn : ARRAY[1..4]OF INT;
	END_STRUCT;
	mnSystem_SignalOut_typ : 	STRUCT
		xOut : ARRAY[1..12]OF BOOL;
		iOut : ARRAY[1..4]OF INT;
	END_STRUCT;
END_TYPE

(*Parameter*)

TYPE
	mnSystemPar_typ : 	STRUCT
		Cfg : mnSystemParCfg_typ;
		Mac : mnSystemParMac_typ;
	END_STRUCT;
	mnSystemParMac_typ : 	STRUCT
		wWarnTemperatureEnvironment : UINT := 750; (*Warnschwelle für Temperaturüberwachung in 0,1 °C*)
	END_STRUCT;
	mnSystemParCfgLine_typ : 	STRUCT
		wModuleID : ARRAY[1..MNSYSTEM_CNT_MODULES]OF UINT;
		sName : ARRAY[1..MNSYSTEM_CNT_MODULES]OF STRING[13];
	END_STRUCT;
	mnSystemParCfg_typ : 	STRUCT
		Lines : ARRAY[1..MNSYSTEM_CNT_MODULELINES]OF mnSystemParCfgLine_typ;
		BindingWarnEnvTemp : ARRAY[1..2]OF mnSystemMdlBinding_typ;
		BindingMotProtCooling : ARRAY[1..2]OF mnSystemMdlBinding_typ;
		BindingOutCooling : ARRAY[1..2]OF mnSystemMdlBinding_typ;
		sSwitchBoxName : ARRAY[1..2]OF STRING[13];
	END_STRUCT;
	mnSystemMdlBinding_typ : 	STRUCT
		wBindIndexModul : UINT; (*Gibt an, welches Modul verwendet wird*)
		wBindIndexChannel : UINT; (* Gibt an, welcher Platz auf dem Modul verwendet wird*)
		sDiscription : STRING[13];
		xInvers : BOOL; (*Invertiertes Eingangssignal*)
	END_STRUCT;
END_TYPE
```

### Pkg_mnSystem.var - Local variables
```iecst
(********************************************************************
 * COPYRIGHT -- Kannegiesser GmbH
 ********************************************************************
 * Program: mnSystem
 * File: mnSystem.var
 * Author: horn
 * Created: January 10, 2012
 ********************************************************************
 * Local variables of program mnSystem
 ********************************************************************)
(*Konstanten*)
VAR CONSTANT
	MNSYSTEM_MSG_BATTERY : UINT := 3;
	MNSYSTEM_MSG_FAN : UINT := 4;
	MNSYSTEM_MSG_ENVTEMP : UINT := 5;
	MNSYSTEM_MSG_WRONGMODULE : UINT := 6;
	MNSYSTEM_MSG_MOTPROTCOOLING : UINT := 7;
END_VAR
(*Variablen*)
VAR
	IFmnSystem : IFmnSystem_typ;
	mnSystemCmd : KG_Cmd_typ;
	mnSystemStat : Stat_typ;
	mnSystemStatAd : mnSystemStatAd_typ;
	mnSystemPar : mnSystemPar_typ;
END_VAR
(*IO*)
VAR
	MDLIn : ARRAY[1..MNSYSTEM_CNT_MODULELINES,1..MNSYSTEM_CNT_MODULES] OF mnSystem_SignalIn_typ;
	MDLOut : ARRAY[1..MNSYSTEM_CNT_MODULELINES,1..MNSYSTEM_CNT_MODULES] OF mnSystem_SignalOut_typ;
END_VAR
```

### mnSystem.History.txt
```
1.00.0	2012-03-16	AH	Neu
1.00.1	2012-03-20 	AH	Abhängigkeiten ergänzt
1.01.0	2012-03-23	AH	Lüfterüberwachung, Temperaturüberwachung
1.02.0	2012-03-23	AH	USB-Stick Überwachung
1.02.1	2012-04-17	AH	Bei unbekannter Modul-ID wird die Modul-ID als CPU-Typ zurückgegeben.
1.03.0	2012-05-11	AH	IO-Variablen eines PowerPanel ergänzt
1.04.0	2012-06-04	AH	USB-Stick-Scan wird sofort nach dem Hochlauf schon einmal durchgeführt. IFmnSystem wurde
						um xUSBStickScanned erweitert.
1.05.0	2012-06-18	AH	CP1584 ergänzt
1.06.0	2012-06-25	AH	Modulüberwachung ergänzt
1.07.0	2012-07-08	AH	Schaltschrankkühlung (2 mögliche Kreise, CPU-Temperatur ist dem 1. Kreis zugeordnet)
						1s- und 500ms-Takt
1.08.0	2012-09-18	AH	CP3484 ergänzt.
```

### CfgMsgStat.mnSystem.txt
```
;****************************
; System Manager
;*****************************
00110, 00003, 00000, 00000;
00110, 00004, 00000, 00000;
00110, 00005, 00000, 00000;
00110, 00006, 00000, 00000;
00110, 00007, 00000, 00000;
```

### Package Logical/Standard/Kanlink/KGFramework/Pkg_mnEth - Ethernet Manager

### Pkg_mnEth.typ - Global data types
```iecst
(********************************************************************
 * COPYRIGHT --
 ********************************************************************
 * File: Global.typ
 * Author: tamme
 * Created: March 17, 2011
 ********************************************************************
 * Global data types of project Ethernetmanagr
 ********************************************************************)

TYPE
	mnEthIP_typ : 	STRUCT
		sIP : STRING[15];
		sGateway : STRING[15];
		sHostname : STRING[15];
		sNetId : STRING[15];
		bNetId1 : USINT;
		bNetId2 : USINT;
		bNetId3 : USINT;
		bRegion : USINT;
		bStation : USINT;
		bNumber : USINT;
	END_STRUCT;
	IFmnEthOut_typ : 	STRUCT
		IP : mnEthIP_typ;
		sEthDevice : STRING[15];
		xDataValid : BOOL;
	END_STRUCT;
	IFmnEthIn_typ : 	STRUCT
		bNodeSwitch : USINT;
	END_STRUCT;
	IFmnEth_typ : 	STRUCT
		In : IFmnEthIn_typ;
		Out : IFmnEthOut_typ;
	END_STRUCT;
	mnEthStatAd_typ : 	STRUCT
		IP : mnEthIP_typ;
		xDataValid : BOOL;
		sPkgVersion : STRING[11];
	END_STRUCT;
	mnEthPar_typ : 	STRUCT
		Cfg : mnEthParCfg_typ;
		Mac : mnEthParMac_typ;
	END_STRUCT;
	mnEthParMac_typ : 	STRUCT
		xStartDHCP : BOOL;
		xStartSNTPClt : BOOL;
		xStartSNTPSrv : BOOL;
		xForceNotSubnetmask : BOOL;
		sIP_SNTP_Srv : STRING[15];
	END_STRUCT;
	mnEthParCfg_typ : 	STRUCT
		bNETid1 : USINT;
		bNETid2 : USINT;
		bNETid3 : USINT;
		bRegion : USINT;
		bStation : USINT;
	END_STRUCT;
END_TYPE
```

### Pkg_mnEth.var - Global variables
```iecst
(********************************************************************
 * COPYRIGHT --
 ********************************************************************
 * File: Global.var
 * Author: tamme
 * Created: March 17, 2011
 ********************************************************************
 * Global variables of project Ethernetmanager
 ********************************************************************)
VAR
	IFmnEth : IFmnEth_typ;
	mnEthPar : mnEthPar_typ;
	mnEthCmd : KG_Cmd_typ;
	mnEthStatAd : mnEthStatAd_typ;
END_VAR
```

### Program Logical/Standard/Kanlink/KGFramework/Pkg_mnEth/mnEth (IEC) - Ethernetmanager

#### mnEthCyclic.st - Cyclic code
```iecst
(********************************************************************
 * COPYRIGHT --
 ********************************************************************
 * Program: mnEth
 * File: mnEthCyclic.st
 * Author: hunholz
 * Created: August 9, 2011
 * Changed: October 7, 2011
 ********************************************************************
 * Implementation of program mnEth
 ********************************************************************)

PROGRAM _CYCLIC

	// Input Messagesystem

	_kgMsgStatus.xAckAva := kgMsgStatus[MNETH_IDX_KGMSGSTAT].xAckAva;
	_kgMsgStatus.xAckFault := kgMsgStatus[MNETH_IDX_KGMSGSTAT].xAckFault;
	_kgMsgStatus.xAckMaint := kgMsgStatus[MNETH_IDX_KGMSGSTAT].xAckMaint;

	_kgMsgStatus.wFunction_ID := 4;

	IF _xmnEthOk THEN

		CASE enEState OF

			es_idle:

				IF _xSetHostname THEN

					enEState := es_SetHostname1;

				ELSIF _xSetDefault THEN

					enEState := es_SetDef1;
					_xCheckedUSB := TRUE;

				ELSIF NOT _xCheckedUSB THEN

					IF IFmnSystem.Out.xUSBStickReady THEN

						enEState := es_SetUSB1;

						_sPathCsv := _sHostname;
						_sPathCsv := CONCAT(_sPathCsv, '\mnEth\mnEth.csv');
						_sDevice := IFmnSystem.Out.sInterfaceUSB;

					END_IF

					_xCheckedUSB := TRUE;

				ELSIF mnEthPar.Mac.xStartDHCP AND IFmnParam.Out.xParamOK AND NOT _xDHCPstarted THEN

					// schaltet den DHCP-Server ein. Nicht dauerhaft. Wird der Maschinenparameter auf FALSE gesetzt
					// dann bleibt der DHCP-Server aus.
					enEState := es_DHCP1;

				ELSIF mnEthPar.Mac.xStartSNTPClt AND IFmnParam.Out.xParamOK AND NOT _xSNTPCltStarted THEN

					enEState := es_SNTPcltStart1;

				ELSIF NOT mnEthPar.Mac.xStartSNTPClt AND IFmnParam.Out.xParamOK AND _xSNTPCltStarted THEN

					enEState := es_SNTPcltStop1;

				ELSIF mnEthPar.Mac.xStartSNTPSrv AND IFmnParam.Out.xParamOK AND NOT _xSNTPSrvStarted THEN

					enEState := es_SNTPsrvStart1;

				ELSIF NOT mnEthPar.Mac.xStartSNTPSrv AND IFmnParam.Out.xParamOK AND _xSNTPSrvStarted THEN

					enEState := es_SNTPsrvStop1;

				ELSIF _bWaitCounter >= 3 THEN

					_xChanged := FALSE;

					_ParSet := _ParAktuell;

					enEState := es_WriteCSV1;

				ELSIF _TONidle.Q THEN

					enEState := es_Change1;

				END_IF

			// Beobachte eingestellte IP und das Gateway
			es_Change1:

				_CfgGetGateway(enable := TRUE, pDevice := ADR(_sEthDevice), pGateway := ADR(_ParGet.Gateway_Adr), Len := SIZEOF(_ParGet.Gateway_Adr));

				IF _CfgGetGateway.status = ERR_OK THEN

					enEState := es_Change2;

				ELSIF _CfgGetGateway.status <> ERR_FUB_BUSY THEN

					_kgMsgStatus.wMsgClass := 11;
					_kgMsgStatus.wMsgNumber := _MNETH_MSG_CHANGE;
					_kgMsgStatus.diMsgAttr1 := UINT_TO_DINT(_CfgGetGateway.status);

					enEState := es_Warning;
				END_IF

			es_Change2:

				_CfgGetIPAddress(enable := TRUE, pDevice := ADR(_sEthDevice), pIPAddr := ADR(_ParGet.IP_Adr), Len := SIZEOF(_ParGet.IP_Adr));

				IF _CfgGetIPAddress.status = ERR_OK THEN

					enEState := es_Change3;

				ELSIF _CfgGetIPAddress.status <> ERR_FUB_BUSY THEN

					_kgMsgStatus.wMsgClass := 11;
					_kgMsgStatus.wMsgNumber := _MNETH_MSG_CHANGE;
					_kgMsgStatus.diMsgAttr1 := UINT_TO_DINT(_CfgGetIPAddress.status);

					enEState := es_Warning;
				END_IF

			es_Change3:

				IF (brsstrcmp(ADR(_ParAktuell.Gateway_Adr), ADR(_ParGet.Gateway_Adr)) = 0)	AND (brsstrcmp(ADR(_ParAktuell.IP_Adr), ADR(_ParGet.IP_Adr)) = 0) THEN

					IF _xChanged THEN

						_bWaitCounter := _bWaitCounter + 1;

					ELSE

						_bWaitCounter := 0;

					END_IF

					enEState := es_idle;

				ELSE

					IF ethInetAton(pIpStr := ADR(_ParGet.IP_Adr), ADR(_lIPAdr)) = ERR_OK THEN

						IF ethInetAton(pIpStr := ADR(_ParGet.Gateway_Adr), ADR(_lGatewayAdr)) = ERR_OK THEN

							_pOctet ACCESS ADR(_lIPAdr);

							_ParGet.IP_ID1 := _pOctet[0];
							_ParGet.IP_ID2 := _pOctet[1];
							_ParGet.IP_ID3 := (_pOctet[2] / 16) * 16;

							_ParGet.Region := _pOctet[2] MOD 16;
							_ParGet.Station := _pOctet[3];

							IF _ParGet.Region = 3 THEN
								_ParGet.Number := kgGetLineNumberW3(Station := _ParGet.Station, pMachineType := ADR(_kgMachineTypeW3));
							ELSE
								_ParGet.Number := 0;
							END_IF

							// NET-Id bestimmen
							_lNetId := _lIPAdr;
							_pOctet ACCESS ADR(_lNetId);

							_pOctet[2] := _ParGet.IP_ID3;
							_pOctet[3] := 0;

							ethInetNtoa(ipAdr := _lNetId, pIpStr := ADR(_ParGet.NetId_Adr));

							_pOctet ACCESS ADR(_lGatewayAdr);

							_ParGet.GWRegion 	:= _pOctet[2] MOD 16;
							_ParGet.GWStation 	:= _pOctet[3];

							enEState := es_Change4;

						END_IF

					END_IF

				END_IF

			es_Change4:

				_CfgSetIPAddr(enable := TRUE, pDevice := ADR(_sEthDevice), pIPAddr := ADR(_ParGet.IP_Adr), Option := cfgOPTION_NON_VOLATILE);

				IF _CfgSetIPAddr.status = ERR_OK THEN

					enEState := es_Change5;

				ELSIF _CfgSetIPAddr.status <> ERR_FUB_BUSY THEN

					_kgMsgStatus.wMsgClass := 11;
					_kgMsgStatus.wMsgNumber := _MNETH_MSG_CHANGE;
					_kgMsgStatus.diMsgAttr1 := UINT_TO_DINT(_CfgSetIPAddr.status);

					enEState := es_Warning;

				END_IF

			es_Change5:

				_CfgSetDefaultGateway(enable := TRUE, pDevice := ADR(_sEthDevice), pGateway := ADR(_ParGet.Gateway_Adr), Option := cfgOPTION_NON_VOLATILE);

				IF _CfgSetDefaultGateway.status = ERR_OK THEN

					enEState := es_Change6;

				ELSIF _CfgSetDefaultGateway.status <> ERR_FUB_BUSY THEN

					_kgMsgStatus.wMsgClass := 11;
					_kgMsgStatus.wMsgNumber := _MNETH_MSG_CHANGE;
					_kgMsgStatus.diMsgAttr1 := UINT_TO_DINT(_CfgSetDefaultGateway.status);

					enEState := es_Warning;

				END_IF

			es_Change6:

				IF NOT mnEthPar.Mac.xForceNotSubnetmask THEN

					_CfgSetSubnetMask(enable := TRUE, pDevice := ADR(_sEthDevice), pSubnetMask := ADR(_sSubnetMask), Option := cfgOPTION_NON_VOLATILE);

					IF _CfgSetSubnetMask.status <> ERR_FUB_BUSY THEN

						enEState := es_Change7;

					END_IF

				ELSE

					enEState := es_Change7;

				END_IF

			es_Change7:

				_pOctet ACCESS ADR(_lBroadcastAdr);

				_pOctet[0] := _ParGet.IP_ID1;
				_pOctet[1] := _ParGet.IP_ID2;
				_pOctet[2] := _ParGet.IP_ID3 + 15;
				_pOctet[3] := 255;

				ethInetNtoa(ADR(_lBroadcastAdr), ADR(_sBroadcastAdr));

				_CfgSetBroadcastAdr(enable := TRUE, pDevice := ADR(_sEthDevice), pBroadcastAddr := ADR(_sBroadcastAdr), Option := cfgOPTION_NON_VOLATILE);

				IF _CfgSetBroadcastAdr.status = ERR_OK THEN

					_ParAktuell := _ParGet;

					_xChanged  := TRUE;

					enEState := es_idle;

				ELSIF _CfgSetBroadcastAdr.status <> ERR_FUB_BUSY THEN

					_kgMsgStatus.wMsgClass := 11;
					_kgMsgStatus.wMsgNumber := _MNETH_MSG_SETDEF;
					_kgMsgStatus.diMsgAttr1 := UINT_TO_DINT(_CfgSetBroadcastAdr.status);

					enEState := es_Warning;

				END_IF

			// Setze Default aus Parameter
			es_SetDef1:

				IF IFmnParam.Out.xParamOK THEN

					_ParSet.IP_ID1 := mnEthPar.Cfg.bNETid1;
					_ParSet.IP_ID2 := mnEthPar.Cfg.bNETid2;
					_ParSet.IP_ID3 := mnEthPar.Cfg.bNETid3;

					_ParSet.Region := mnEthPar.Cfg.bRegion;
					_ParSet.Station := mnEthPar.Cfg.bStation;

					_ParSet.GWRegion 	:= 15;
					_ParSet.GWStation 	:= 254;

					IF _ParAktuell.Region = 3 THEN
						_ParSet.Number := kgGetLineNumberW3(Station := _ParSet.Station, pMachineType := ADR(_kgMachineTypeW3));
					ELSE
						_ParSet.Number := 0;
					END_IF

					_pOctet ACCESS ADR(_lIPAdr);

					_pOctet[0] := _ParSet.IP_ID1;
					_pOctet[1] := _ParSet.IP_ID2;
					_pOctet[2] := _ParSet.IP_ID3 + _ParSet.Region;
					_pOctet[3] := _ParSet.Station;

					ethInetNtoa(_lIPAdr, ADR(_ParSet.IP_Adr));

					// NET-Id bestimmen
					_lNetId := _lIPAdr;
					_pOctet ACCESS ADR(_lNetId);

					_pOctet[2] := _ParSet.IP_ID3;
					_pOctet[3] := 0;

					ethInetNtoa(ipAdr := _lNetId, pIpStr := ADR(_ParSet.NetId_Adr));

					// Gateway Adress
					_pOctet[0] := _ParSet.IP_ID1;
					_pOctet[1] := _ParSet.IP_ID2;
					_pOctet[2] := _ParSet.IP_ID3 + _ParSet.GWRegion;
					_pOctet[3] := _ParSet.GWStation;

					ethInetNtoa(_lIPAdr, ADR(_ParSet.Gateway_Adr));

					enEState := es_SetDef2;

				END_IF

			es_SetDef2:

				_CfgSetIPAddr(enable := TRUE, pDevice := ADR(_sEthDevice), pIPAddr := ADR(_ParSet.IP_Adr), Option := cfgOPTION_VOLATILE);

				IF _CfgSetIPAddr.status = ERR_OK THEN

					enEState := es_SetDef3;

				ELSIF _CfgSetIPAddr.status <> ERR_FUB_BUSY THEN

					_kgMsgStatus.wMsgClass := 11;
					_kgMsgStatus.wMsgNumber := _MNETH_MSG_SETDEF;
					_kgMsgStatus.diMsgAttr1 := UINT_TO_DINT(_CfgSetIPAddr.status);

					_xSetDefault := FALSE;
					enEState := es_Warning;

				END_IF

			es_SetDef3:

				_CfgGetGateway(enable := TRUE, pDevice := ADR(_sEthDevice), pGateway := ADR(_ParSet.Gateway_Adr), Len := SIZEOF(_ParSet.Gateway_Adr));

				IF _CfgGetGateway.status = ERR_OK THEN

					enEState := es_SetDef4;

				ELSIF _CfgGetGateway.status <> ERR_FUB_BUSY THEN

					_kgMsgStatus.wMsgClass := 11;
					_kgMsgStatus.wMsgNumber := _MNETH_MSG_SETDEF;
					_kgMsgStatus.diMsgAttr1 := UINT_TO_DINT(_CfgGetGateway.status);

					_xSetDefault := FALSE;
					enEState := es_Warning;

				END_IF

			es_SetDef4:

				IF NOT mnEthPar.Mac.xForceNotSubnetmask THEN

					_CfgSetSubnetMask(enable := TRUE, pDevice := ADR(_sEthDevice), pSubnetMask := ADR(_sSubnetMask), Option := cfgOPTION_VOLATILE);

					IF _CfgSetSubnetMask.status <> ERR_FUB_BUSY THEN

						enEState := es_SetDef5;

					END_IF

				ELSE

					enEState := es_SetDef5;

				END_IF

			es_SetDef5:

				_pOctet ACCESS ADR(_lBroadcastAdr);

				_pOctet[0] := _ParSet.IP_ID1;
				_pOctet[1] := _ParSet.IP_ID2;
				_pOctet[2] := _ParSet.IP_ID3 + 15;
				_pOctet[3] := 255;

				ethInetNtoa(ADR(_lBroadcastAdr), ADR(_sBroadcastAdr));

				_CfgSetBroadcastAdr(enable := TRUE, pDevice := ADR(_sEthDevice), pBroadcastAddr := ADR(_sBroadcastAdr), Option := cfgOPTION_VOLATILE);

				IF _CfgSetBroadcastAdr.status = ERR_OK THEN

					_xSetDefault := FALSE;
					enEState := es_WriteCSV1;

				ELSIF _CfgSetBroadcastAdr.status <> ERR_FUB_BUSY THEN

					_kgMsgStatus.wMsgClass := 11;
					_kgMsgStatus.wMsgNumber := _MNETH_MSG_SETDEF;
					_kgMsgStatus.diMsgAttr1 := UINT_TO_DINT(_CfgSetBroadcastAdr.status);

					_xSetDefault := FALSE;
					enEState := es_Warning;

				END_IF

			es_SetUSB1:

				_FileOpenCsv(enable := TRUE, pDevice := ADR(_sDevice), pFile := ADR(_sPathCsv), mode := fiREAD_ONLY);

				IF _FileOpenCsv.status = ERR_OK THEN

					enEState := es_SetUSB2;

				ELSE

					enEState := es_idle;

				END_IF

			es_SetUSB2:

				_FileReadCsv(enable := TRUE, ident := _FileOpenCsv.ident, pDest := _pParseMem, len := 256);

				IF _FileReadCsv.status = ERR_OK THEN

					_GetCsvDat.enable := TRUE;
					brwcsncpy( ADR(_GetCsvDat.utfCsvString), _pParseMem+2, 126);
					_GetCsvDat();

					IF _GetCsvDat.RowType = 90 THEN

						_ParSet.IP_Adr := WSTRING_TO_STRING(_GetCsvDat.CsvIPRow.utfIP_Adress);
						_ParSet.Gateway_Adr := WSTRING_TO_STRING(_GetCsvDat.CsvIPRow.utfGateway);

						IF ethInetAton(pIpStr := ADR(_ParSet.IP_Adr), ADR(_lIPAdr)) = ERR_OK THEN

							IF ethInetAton(pIpStr := ADR(_ParSet.Gateway_Adr), ADR(_lGatewayAdr)) = ERR_OK THEN

								_pOctet ACCESS ADR(_lIPAdr);

								_ParSet.IP_ID1 := _pOctet[0];
								_ParSet.IP_ID2 := _pOctet[1];
								_ParSet.IP_ID3 := (_pOctet[2] / 16) * 16;

								_ParSet.Region := _pOctet[2] MOD 16;
								_ParSet.Station := _pOctet[3];

								IF _ParSet.Region = 3 THEN
									_ParSet.Number := kgGetLineNumberW3(Station := _ParSet.Station, pMachineType := ADR(_kgMachineTypeW3));
								ELSE
									_ParSet.Number := 0;
								END_IF

								// NET-Id bestimmen
								_lNetId := _lIPAdr;
								_pOctet ACCESS ADR(_lNetId);

								_pOctet[2] := _ParSet.IP_ID3;
								_pOctet[3] := 0;

								ethInetNtoa(ipAdr := _lNetId, pIpStr := ADR(_ParSet.NetId_Adr));

								_pOctet ACCESS ADR(_lGatewayAdr);

								_ParSet.GWRegion := _pOctet[2] MOD 16;
								_ParSet.GWStation := _pOctet[3];

								enEState := es_SetUSB3;

							END_IF

						END_IF

					END_IF

				END_IF

			es_SetUSB3:

				_CfgSetIPAddr(enable := TRUE, pDevice := ADR(_sEthDevice), pIPAddr := ADR(_ParSet.IP_Adr), Option := cfgOPTION_VOLATILE);

				IF _CfgSetIPAddr.status = ERR_OK THEN

					enEState := es_SetUSB4;

				ELSIF _CfgSetIPAddr.status <> ERR_FUB_BUSY THEN

					_kgMsgStatus.wMsgClass := 11;
					_kgMsgStatus.wMsgNumber := _MNETH_MSG_SETUSB;
					_kgMsgStatus.diMsgAttr1 := UINT_TO_DINT(_CfgSetIPAddr.status);

					_xSetDefault := FALSE;
					enEState := es_Warning;

				END_IF

			es_SetUSB4:

				_CfgGetGateway(enable := TRUE, pDevice := ADR(_sEthDevice), pGateway := ADR(_ParSet.Gateway_Adr), Len := SIZEOF(_ParSet.Gateway_Adr));

				IF _CfgGetGateway.status = ERR_OK THEN

					enEState := es_SetUSB5;

				ELSIF _CfgGetGateway.status <> ERR_FUB_BUSY THEN

					_kgMsgStatus.wMsgClass := 11;
					_kgMsgStatus.wMsgNumber := _MNETH_MSG_SETUSB;
					_kgMsgStatus.diMsgAttr1 := UINT_TO_DINT(_CfgGetGateway.status);

					_xSetDefault := FALSE;
					enEState := es_Warning;

				END_IF

			es_SetUSB5:

				IF NOT mnEthPar.Mac.xForceNotSubnetmask THEN

					_CfgSetSubnetMask(enable := TRUE, pDevice := ADR(_sEthDevice), pSubnetMask := ADR(_sSubnetMask), Option := cfgOPTION_VOLATILE);

					IF _CfgSetSubnetMask.status <> ERR_FUB_BUSY THEN

						enEState := es_SetUSB6;

					END_IF

				ELSE

					enEState := es_SetUSB6;

				END_IF

			es_SetUSB6:

				_pOctet ACCESS ADR(_lBroadcastAdr);

				_pOctet[0] := _ParSet.IP_ID1;
				_pOctet[1] := _ParSet.IP_ID2;
				_pOctet[2] := _ParSet.IP_ID3 + 15;
				_pOctet[3] := 255;

				ethInetNtoa(ADR(_lBroadcastAdr), ADR(_sBroadcastAdr));

				_CfgSetBroadcastAdr(enable := TRUE, pDevice := ADR(_sEthDevice), pBroadcastAddr := ADR(_sBroadcastAdr), Option := cfgOPTION_VOLATILE);

				IF _CfgSetBroadcastAdr.status = ERR_OK THEN

					_xSetDefault := FALSE;
					enEState := es_WriteCSV1;

				ELSIF _CfgSetBroadcastAdr.status <> ERR_FUB_BUSY THEN

					_kgMsgStatus.wMsgClass := 11;
					_kgMsgStatus.wMsgNumber := _MNETH_MSG_SETUSB;
					_kgMsgStatus.diMsgAttr1 := UINT_TO_DINT(_CfgSetBroadcastAdr.status);

					_xSetDefault := FALSE;
					enEState := es_Warning;

				END_IF

			es_WriteCSV1:

				_ParAktuell := _ParSet;

				brsmemset(_pParseMem, 0, 256);

				_lFileSize := 0;

				brwcsconv(ADR( _IPRow.utfIP_Adress), ADR(_ParSet.IP_Adr), 0);
				brwcsconv(ADR(_IPRow.utfGateway), ADR(_ParSet.Gateway_Adr), 0);

				_WriteBOM(enable := TRUE, pMem := _pParseMem, lMaxSize := 256, lSize := _lFileSize);
				_WriteCsv90(enable := TRUE, pMem := _pParseMem, lMaxSize := 256, IPRow := _IPRow, lSize := _lFileSize);

				enEState := es_WriteCSV2;

			es_WriteCSV2:

				_FileDeleteCsv(enable := TRUE, pDevice := ADR(KG_DEVICE_COMPACTFLASH), pName := ADR(_sPathCsv));

				IF _FileDeleteCsv.status <> ERR_FUB_BUSY THEN

					enEState := es_WriteCSV3;

				END_IF

			es_WriteCSV3:

				_FileCreateCsv(enable := TRUE, pDevice := ADR(KG_DEVICE_COMPACTFLASH), pFile := ADR(_sPathCsv));

				IF _FileCreateCsv.status = ERR_OK THEN

					enEState := es_WriteCSV5;

				ELSIF _FileCreateCsv.status <> ERR_FUB_BUSY THEN

					_kgMsgStatus.wMsgClass := 11;
					_kgMsgStatus.wMsgNumber := _MNETH_MSG_WRITECSV;
					_kgMsgStatus.diMsgAttr1 := UINT_TO_DINT(_FileCreateCsv.status);

					enEState := es_Warning;

				END_IF

			es_WriteCSV4:

				_FileOpenCsv(enable := TRUE, pDevice := ADR(KG_DEVICE_COMPACTFLASH), pFile := ADR(_sPathCsv), mode := fiWRITE_ONLY);

				IF _FileOpenCsv.status = ERR_OK THEN

					enEState := es_WriteCSV5;

				ELSIF _FileOpenCsv.status <> ERR_FUB_BUSY THEN

					_kgMsgStatus.wMsgClass := 11;
					_kgMsgStatus.wMsgNumber := _MNETH_MSG_WRITECSV;
					_kgMsgStatus.diMsgAttr1 := UINT_TO_DINT(_FileOpenCsv.status);

					enEState := es_Warning;

				END_IF

			es_WriteCSV5:

				_FileWriteCsv(enable := TRUE, ident := _FileCreateCsv.ident, offset := 0, pSrc := _pParseMem, len := _lFileSize);

				IF _FileWriteCsv.status <> ERR_FUB_BUSY THEN

					enEState := es_WriteCSV6;

				END_IF

			es_WriteCSV6:

				_FileCloseCsv(enable := TRUE, ident := _FileCreateCsv.ident);

				IF _FileCloseCsv.status <> ERR_FUB_BUSY THEN

					_bWaitCounter := 0;
					_xChanged := FALSE;

					enEState := es_idle;

				END_IF

			es_Warning:

				_bWaitCounter := 0;
				_xChanged := FALSE;

				IF _TONwarning.Q THEN

					brsmemset(ADR(_kgMsgStatus),0,SIZEOF(kgMsgStatus[0]));
					_kgMsgStatus.wFunction_ID := 4;

					enEState := es_idle;

				END_IF

			es_DHCP1:

				brsstrcpy(ADR(_cfgLease.name), ADR('KANLINK'));
				brsstrcpy(ADR(_cfgLease.defaultGateway), ADR(_ParAktuell.Gateway_Adr));
				brsstrcpy(ADR(_cfgLease.subnetMask), ADR(_sSubnetMask));

				// Startadresse
				_lIPAdr := 0;
				_pOctet ACCESS ADR(_lIPAdr);
				_pOctet[0] := _ParAktuell.IP_ID1;
				_pOctet[1] := _ParAktuell.IP_ID2;
				_pOctet[2] := _ParAktuell.IP_ID3;

				_pOctet[3] := 150;

				ethInetNtoa(_lIPAdr, ADR(_cfgLease.startAdr));

				// Stopadresse
				_pOctet[3] := 169;

				ethInetNtoa(_lIPAdr, ADR(_cfgLease.stopAdr));

				_cfgLease.leaseTimeout := -1;

				enEState := es_DHCP2;

			es_DHCP2:

				_CfgSetDhcpsData(enable := TRUE, pInterfaceList := ADR(_sEthDevice), pLeases := ADR(_cfgLease), numLeases := 1, option := cfgOPTION_VOLATILE);

				IF (_CfgSetDhcpsData.status = ERR_OK) THEN

					enEState := es_DHCP3;

				ELSIF _CfgSetDhcpsData.status <> ERR_FUB_BUSY THEN

					enEState := es_idle;
					_xDHCPstarted := TRUE;

				END_IF

			es_DHCP3:

				_CfgSetDhcpServer(enable := TRUE, start := 1, option := cfgOPTION_VOLATILE);

				IF _CfgSetDhcpServer.status <> ERR_FUB_BUSY THEN

					enEState := es_idle;
					_xDHCPstarted := TRUE;

				END_IF

			es_SNTPcltStart1:

				_CfgSetSntpClient(enable := TRUE, run := 1, pServerAddr := ADR(mnEthPar.Mac.sIP_SNTP_Srv), sntpcInterval := 30, rtcInterval := 30, option := cfgOPTION_VOLATILE);

				IF _CfgSetSntpClient.status <> ERR_FUB_BUSY THEN

					enEState := es_idle;
					_xSNTPCltStarted := TRUE;

				END_IF

			es_SNTPcltStop1:

				_CfgSetSntpClient(enable := TRUE, run := 0, pServerAddr := ADR(mnEthPar.Mac.sIP_SNTP_Srv), sntpcInterval := 30, rtcInterval := 30, option := cfgOPTION_VOLATILE);

				IF _CfgSetSntpClient.status <> ERR_FUB_BUSY THEN

					enEState := es_idle;
					_xSNTPCltStarted := FALSE;

				END_IF

			es_SNTPsrvStart1:

				_CfgSetSntpServer(enable := TRUE, start := 1, option := cfgOPTION_VOLATILE);

				IF _CfgSetSntpServer.status <> ERR_FUB_BUSY THEN

					enEState := es_idle;
					_xSNTPSrvStarted := TRUE;

				END_IF

			es_SNTPsrvStop1:

				_CfgSetSntpServer(enable := TRUE, start := 0, option := cfgOPTION_VOLATILE);

				IF _CfgSetSntpServer.status <> ERR_FUB_BUSY THEN

					enEState := es_idle;
					_xSNTPSrvStarted := FALSE;

				END_IF

			es_SetHostname1:

				IF IFmnParam.Out.xParamOK THEN

					brwcsconv(ADR(_sMnr), ADR(IFmnParam.Out.utfMachineNumber) ,1);

					_sHostname := 'KaMa';
					brsstrcat(ADR(_sHostname), ADR(_sMnr));

					enEState := es_SetHostname2;

				END_IF

			es_SetHostname2:

				_CfgGetHostName(enable := TRUE, pHostName := ADR(_sActHostname), Len := SIZEOF(_sActHostname));

				IF _CfgGetHostName.status = ERR_OK THEN

					IF brsstrcmp(ADR(_sHostname), ADR(_sActHostname)) = 0 THEN

						_xSetHostname := FALSE;
						enEState := es_idle;

					ELSE

						enEState := es_SetHostname3;

					END_IF

				ELSIF _CfgGetHostName.status <> ERR_FUB_BUSY THEN

					_xSetHostname := FALSE;
					enEState := es_idle;

				END_IF

			es_SetHostname3:

				_CfgSetHostName(enable := TRUE, pHostName := ADR(_sHostname), Option := cfgOPTION_NON_VOLATILE);

				IF _CfgSetHostName.status <> ERR_FUB_BUSY THEN

					_xSetHostname := FALSE;
					enEState := es_idle;

				END_IF

		END_CASE

		_TONidle(IN := enEState = es_idle, PT := T#2s);

		_TONwarning(IN := enEState = es_Warning, PT := T#30s);

		// Ethernetdaten übergeben
		mnEthStatAd.IP.sHostname		:= _sHostname;
		mnEthStatAd.IP.sIP 				:= _ParAktuell.IP_Adr;
		mnEthStatAd.IP.sGateway 		:= _ParAktuell.Gateway_Adr;
		mnEthStatAd.IP.sNetId			:= _ParAktuell.NetId_Adr;
		mnEthStatAd.IP.bNetId1			:= _ParAktuell.IP_ID1;
		mnEthStatAd.IP.bNetId2			:= _ParAktuell.IP_ID2;
		mnEthStatAd.IP.bNetId3			:= _ParAktuell.IP_ID3;
		mnEthStatAd.IP.bNumber			:= _ParAktuell.Number;
		mnEthStatAd.IP.bRegion			:= _ParAktuell.Region;
		mnEthStatAd.IP.bStation			:= _ParAktuell.Station;
		IFmnEth.Out.IP					:= mnEthStatAd.IP;
		IFmnEth.Out.sEthDevice 			:= _sEthDevice;
		mnEthStatAd.xDataValid			:= NOT _xSetDefault AND NOT _xSetHostname;
		IFmnEth.Out.xDataValid			:= mnEthStatAd.xDataValid;

	ELSE

		_kgMsgStatus.wMsgClass := 11;

		mnEthStatAd.xDataValid := FALSE;

	END_IF // _xmnEthOk

	// MsgSystem Output

	IF NOT IFmnTest.Out.xNoMessages THEN

		kgMsgStatus[MNETH_IDX_KGMSGSTAT].diMaintAttr1 		:= _kgMsgStatus.diMaintAttr1;
		kgMsgStatus[MNETH_IDX_KGMSGSTAT].diMaintAttr2 		:= _kgMsgStatus.diMaintAttr2;
		kgMsgStatus[MNETH_IDX_KGMSGSTAT].diMsgAttr1 		:= _kgMsgStatus.diMsgAttr1;
		kgMsgStatus[MNETH_IDX_KGMSGSTAT].diMsgAttr2 		:= _kgMsgStatus.diMsgAttr2;
		kgMsgStatus[MNETH_IDX_KGMSGSTAT].sMaintAttrTxt 		:= _kgMsgStatus.sMaintAttrTxt;
		kgMsgStatus[MNETH_IDX_KGMSGSTAT].sMsgAttrTxt		:= _kgMsgStatus.sMsgAttrTxt;
		kgMsgStatus[MNETH_IDX_KGMSGSTAT].wFunction_ID		:= _kgMsgStatus.wFunction_ID;
		kgMsgStatus[MNETH_IDX_KGMSGSTAT].wInstance			:= _kgMsgStatus.wInstance;
		kgMsgStatus[MNETH_IDX_KGMSGSTAT].wMaintAckLevel		:= _kgMsgStatus.wMaintAckLevel;
		kgMsgStatus[MNETH_IDX_KGMSGSTAT].wMaintNumber		:= _kgMsgStatus.wMaintNumber;
		kgMsgStatus[MNETH_IDX_KGMSGSTAT].wMsgAckLevel		:= _kgMsgStatus.wMsgAckLevel;
		kgMsgStatus[MNETH_IDX_KGMSGSTAT].wMsgClass			:= _kgMsgStatus.wMsgClass;
		kgMsgStatus[MNETH_IDX_KGMSGSTAT].wMsgNumber			:= _kgMsgStatus.wMsgNumber;
		kgMsgStatus[MNETH_IDX_KGMSGSTAT].xAckRead			:= _kgMsgStatus.xAckRead;

	END_IF

END_PROGRAM
```

#### mnEthInit.st - Initialization code
```iecst
(********************************************************************
 * COPYRIGHT --
 ********************************************************************
 * Program: mnEth
 * File: mnEthInit.st
 * Author: hunholz
 * Created: August 9, 2011
 * Changed: February 3, 2012 2.07.0
 ********************************************************************
 * Implementation of program mnEth
 ********************************************************************)

PROGRAM _INIT

	_xmnEthOk := TRUE;

	_xDHCPstarted := FALSE;
	_xSNTPSrvStarted := FALSE;
	_xSNTPCltStarted := FALSE;

	brsmemset(ADR(kgMsgStatus[MNETH_IDX_KGMSGSTAT]),0,SIZEOF(kgMsgStatus[0]));

	kgMsgStatus[MNETH_IDX_KGMSGSTAT].wFunction_ID := 4;

	// Packet-Version auslesen mit MO_ver aus SYS_lib und für den Additional Status zur Verfügung stellen

	_sPkgName := 'mnEth';

	IF ( MO_ver(ADR(_sPkgName), 0, ADR(_VerStruc)) = 0 ) THEN

		brsmemcpy(ADR(mnEthStatAd.sPkgVersion), ADR(_VerStruc.version), SIZEOF(_VerStruc.version));

	ELSE

		mnEthStatAd.sPkgVersion := '---';

	END_IF

	//***********************************************
	//Lese das Ethernet-Device der CPU aus
	//***********************************************
	REPEAT

		_GetEthPort(enable := TRUE, adrIF := ADR(_sEthDevice));

	UNTIL

		_GetEthPort.status <> ERR_FUB_BUSY

	END_REPEAT

	IFmnEth.Out.sEthDevice := _sEthDevice;

	IF brsstrcmp(ADR(_sEthDevice), ADR('ERR')) = 0 THEN

		kgMsgStatus[MNETH_IDX_KGMSGSTAT].wMsgAckLevel := 0;
		kgMsgStatus[MNETH_IDX_KGMSGSTAT].wMsgClass := 10;
		kgMsgStatus[MNETH_IDX_KGMSGSTAT].wMsgNumber := _MNETH_MSG_IFDEVICE;

		_xmnEthOk := FALSE;

	END_IF

	//**********************************************************
	//Bestimme den Hostnamen der SPS und setze ihn
	//**********************************************************

	_xSetDefault := FALSE;

	IF IFmnEth.In.bNodeSwitch = 16#FE THEN

		// Setze auf jeden Fall die Default Adresse
		_xSetDefault := TRUE;

	END_IF

	//********************************************************************************************
	//Erzeuge einen Speicherbereich zum parsen oder schreiben von CSV-Dateien
	//********************************************************************************************

	_pParseMem := 0;

	_MemPartCreate(enable := TRUE, len := 512);

	IF _MemPartCreate.status = ERR_OK THEN

		_MemPartAlloc(enable := TRUE, ident := _MemPartCreate.ident, len := 256);

		IF _MemPartAlloc.status = ERR_OK THEN

			_pParseMem := _MemPartAlloc.mem;

		ELSE

			kgMsgStatus[MNETH_IDX_KGMSGSTAT].wMsgAckLevel := 0;
			kgMsgStatus[MNETH_IDX_KGMSGSTAT].wMsgClass := 10;
			kgMsgStatus[MNETH_IDX_KGMSGSTAT].wMsgNumber := _MNETH_MSG_MEM;

			_xmnEthOk := FALSE;

		END_IF

	ELSE

		kgMsgStatus[MNETH_IDX_KGMSGSTAT].wMsgAckLevel := 0;
		kgMsgStatus[MNETH_IDX_KGMSGSTAT].wMsgClass := 10;
		kgMsgStatus[MNETH_IDX_KGMSGSTAT].wMsgNumber := _MNETH_MSG_MEM;

		_xmnEthOk := FALSE;

	END_IF

	//********************************************************************************
	// Sicherstellen, dass das Verzeichnis mnEth auf der CF-Card existiert
	//********************************************************************************

	_DirInfo(enable := TRUE, pDevice := ADR(KG_DEVICE_COMPACTFLASH), pPath := ADR('mnEth'));

	IF _DirInfo.status <> ERR_OK THEN

		_DirCreate(enable := TRUE, pDevice := ADR(KG_DEVICE_COMPACTFLASH), pName := ADR('mnEth'));

	END_IF

	//*****************************************************************************************************
	// Wenn nicht default gesetzt werden soll, csv-Datei auf CF suchen
	//*****************************************************************************************************

	_xSetIPFromCF := FALSE;

	_sPathCsv := 'mnEth\mnEth.csv';

	IF _xmnEthOk THEN

		IF NOT _xSetDefault THEN

			_sPathCsv := 'mnEth\mnEth.csv';

			_FileOpenCsv(enable := TRUE, pDevice := ADR(KG_DEVICE_COMPACTFLASH), pFile := ADR(_sPathCsv), mode := fiREAD_ONLY);

			IF _FileOpenCsv.status = ERR_OK THEN

				_FileReadCsv(enable := TRUE, ident := _FileOpenCsv.ident, pDest := _pParseMem, len := 256);

				IF _FileReadCsv.status = ERR_OK THEN

					_GetCsvDat.enable := TRUE;
					brwcsncpy( ADR(_GetCsvDat.utfCsvString), _pParseMem+2, 126);
					// Nur erste Zeile
					_lPosLF := brwcschr(ADR(_GetCsvDat.utfCsvString),16#0A);
					_lPosCR := brwcschr(ADR(_GetCsvDat.utfCsvString),16#0D);
					IF (_lPosCR <> 0) THEN
						brsmemset(_lPosCR , 0, 2);
					END_IF
					IF (_lPosLF <> 0) THEN
						brsmemset(_lPosLF , 0, 2);
					END_IF

					_GetCsvDat();

					IF _GetCsvDat.RowType = 90 THEN

						brwcsconv(ADR(_ParSetCF.IP_Adr), ADR(_GetCsvDat.CsvIPRow.utfIP_Adress), 1);
						brwcsconv(ADR(_ParSetCF.Gateway_Adr), ADR( _GetCsvDat.CsvIPRow.utfGateway), 1);

						IF ethInetAton(pIpStr := ADR(_ParSetCF.IP_Adr), ADR(_lIPAdr)) = ERR_OK THEN

							IF ethInetAton(pIpStr := ADR(_ParSetCF.Gateway_Adr), ADR(_lGatewayAdr)) = ERR_OK THEN

								_pOctet ACCESS ADR(_lIPAdr);

								_ParSetCF.IP_ID1 := _pOctet[0];
								_ParSetCF.IP_ID2 := _pOctet[1];
								_ParSetCF.IP_ID3 := (_pOctet[2] / 16) * 16;

								_ParSetCF.Region := _pOctet[2] MOD 16;
								_ParSetCF.Station := _pOctet[3];

								IF _ParSetCF.Region = 3 THEN
									_ParSetCF.Number := kgGetLineNumberW3(Station := _ParSetCF.Station, pMachineType := ADR(_kgMachineTypeW3));
								ELSE
									_ParSetCF.Number := 0;
								END_IF

								// NET-Id bestimmen
								_lNetId := _lIPAdr;
								_pOctet ACCESS ADR(_lNetId);

								_pOctet[2] := _ParSetCF.IP_ID3;
								_pOctet[3] := 0;

								ethInetNtoa(ipAdr := _lNetId, pIpStr := ADR(_ParSetCF.NetId_Adr));

								_pOctet ACCESS ADR(_lGatewayAdr);

								_ParSetCF.GWRegion 	:= _pOctet[2] MOD 16;
								_ParSetCF.GWStation := _pOctet[3];

								_xSetIPFromCF := TRUE;

							END_IF

						END_IF

					END_IF

				END_IF

				_FileCloseCsv(enable := TRUE, ident := _FileOpenCsv.ident);

			END_IF

		END_IF

	END_IF

	//*****************************************************************************************************
	// Adressen von CF setzen
	//*****************************************************************************************************

	IF _xmnEthOk THEN

		IF _xSetIPFromCF THEN

			_ParSet := _ParSetCF;

			// Für Testzwecke in Hausnetzen mit anderer Netzwerkmaske

//			#ifndef NoSubnetMask
//
//			_CfgGetSubnetMask(enable := TRUE, pDevice := ADR(_sEthDevice), pSubnetMask := ADR(_sActSubnetMask), Len := SIZEOF(_sActSubnetMask));
//
//			IF (brsstrcmp(ADR(_sActSubnetMask), ADR(_sSubnetMask)) <> 0) THEN
//
//				_CfgSetSubnetMask(enable := TRUE, pDevice := ADR(_sEthDevice), pSubnetMask := ADR(_sSubnetMask), Option := cfgOPTION_NON_VOLATILE);
//
//			END_IF
//			#endif

			_pOctet ACCESS ADR(_lBroadcastAdr);

			_pOctet[0] := _ParSet.IP_ID1;
			_pOctet[1] := _ParSet.IP_ID2;
			_pOctet[2] := _ParSet.IP_ID3 + 15;
			_pOctet[3] := 255;

			ethInetNtoa(ADR(_lBroadcastAdr), ADR(_sBroadcastAdr));

			_CfgGetBroadcastAdr(enable := TRUE, pDevice := ADR(_sEthDevice), pBroadcastAddr := ADR(_sActBroadcastAdr), Len := SIZEOF(_sActBroadcastAdr));

			IF (brsstrcmp(ADR(_sActBroadcastAdr), ADR(_sBroadcastAdr)) <> 0) THEN

				_CfgSetBroadcastAdr(enable := TRUE, pDevice := ADR(_sEthDevice), pBroadcastAddr := ADR(_sBroadcastAdr), Option := cfgOPTION_NON_VOLATILE);

			END_IF

			_CfgGetIPAddress(enable := TRUE, pDevice := ADR(_sEthDevice), pIPAddr := ADR(_sActIPAdr), Len := SIZEOF(_sActIPAdr));

			IF (brsstrcmp(ADR(_sActIPAdr), ADR(_ParSet.IP_Adr)) <> 0) THEN

				_CfgSetIPAddr(enable := TRUE, pDevice := ADR(_sEthDevice), pIPAddr := ADR(_ParSet.IP_Adr), Option := cfgOPTION_NON_VOLATILE);

			END_IF

			_CfgGetGateway(enable := TRUE, pDevice := ADR(_sEthDevice), pGateway := ADR(_sActGateway), Len := SIZEOF(_sActGateway));

			IF (brsstrcmp(ADR(_sActGateway), ADR(_ParSet.Gateway_Adr)) <> 0) THEN

				_CfgSetDefaultGateway(enable := TRUE, pDevice := ADR(_sEthDevice), pGateway := ADR(_ParSet.Gateway_Adr), Option := cfgOPTION_NON_VOLATILE);

			END_IF

			_ParAktuell := _ParSet;

		ELSE

			_CfgGetGateway(enable := TRUE, pDevice := ADR(_sEthDevice), pGateway := ADR(_ParAktuell.Gateway_Adr), Len := SIZEOF(_ParAktuell.Gateway_Adr));

			_CfgGetIPAddress(enable := TRUE, pDevice := ADR(_sEthDevice), pIPAddr := ADR(_ParAktuell.IP_Adr), Len := SIZEOF(_ParAktuell.IP_Adr));

			IF ethInetAton(pIpStr := ADR(_ParAktuell.IP_Adr), ADR(_lIPAdr)) = ERR_OK THEN

				IF ethInetAton(pIpStr := ADR(_ParAktuell.Gateway_Adr), ADR(_lGatewayAdr)) = ERR_OK THEN

					_pOctet ACCESS ADR(_lIPAdr);

					_ParAktuell.IP_ID1 := _pOctet[0];
					_ParAktuell.IP_ID2 := _pOctet[1];
					_ParAktuell.IP_ID3 := (_pOctet[2] / 16) * 16;

					_ParAktuell.Region := _pOctet[2] MOD 16;
					_ParAktuell.Station := _pOctet[3];

					IF _ParAktuell.Region = 3 THEN
						_ParAktuell.Number := kgGetLineNumberW3(Station := _ParAktuell.Station, pMachineType := ADR(_kgMachineTypeW3));
					ELSE
						_ParAktuell.Number := 0;
					END_IF

					// NET-Id bestimmen
					_lNetId := _lIPAdr;
					_pOctet ACCESS ADR(_lNetId);

					_pOctet[2] := _ParAktuell.IP_ID3;
					_pOctet[3] := 0;

					ethInetNtoa(ipAdr := _lNetId, pIpStr := ADR(_ParAktuell.NetId_Adr));

					_pOctet ACCESS ADR(_lGatewayAdr);

					_ParAktuell.GWRegion 	:= _pOctet[2] MOD 16;
					_ParAktuell.GWStation 	:= _pOctet[3];

				END_IF

			END_IF

		END_IF

		_xChanged := FALSE;

	END_IF

END_PROGRAM
```

#### mnEth.typ - Local data types
```iecst
(********************************************************************
 * COPYRIGHT --
 ********************************************************************
 * Program: mnEth
 * File: mnEth.typ
 * Author: tamme
 * Created: March 17, 2011
 ********************************************************************
 * Local data types of program mnEth
 ********************************************************************)

TYPE
	enumEthernetState :
		(
		es_idle := 0,
		es_SetDef1 := 100,
		es_SetDef2,
		es_SetDef3,
		es_SetDef4,
		es_SetDef5,
		es_WriteCSV1 := 200,
		es_WriteCSV2,
		es_WriteCSV3,
		es_WriteCSV4,
		es_WriteCSV5,
		es_WriteCSV6,
		es_Change1 := 300,
		es_Change2,
		es_Change3,
		es_Change4,
		es_Change5,
		es_Change6,
		es_Change7,
		es_DHCP1 := 400,
		es_DHCP2,
		es_DHCP3,
		es_SNTPcltStart1 := 500,
		es_SNTPcltStop1 := 510,
		es_SNTPsrvStart1 := 520,
		es_SNTPsrvStop1 := 530,
		es_SetHostname1 := 600,
		es_SetHostname2,
		es_SetHostname3,
		es_SetUSB1 := 700,
		es_SetUSB2,
		es_SetUSB3,
		es_SetUSB4,
		es_SetUSB5,
		es_SetUSB6,
		es_Warning := 900
		);
	_EthPar_typ : 	STRUCT
		IP_ID1 : USINT;
		IP_ID2 : USINT;
		IP_ID3 : USINT;
		Region : USINT;
		Station : USINT;
		Number : USINT;
		GWRegion : USINT;
		GWStation : USINT;
		IP_Adr : STRING[15];
		Gateway_Adr : STRING[15];
		NetId_Adr : STRING[15];
	END_STRUCT;
END_TYPE
```

#### mnEth.var - Local variables
```iecst
(********************************************************************
 * COPYRIGHT --
 ********************************************************************
 * Program: mnEth
 * File: mnEth.var
 * Author: tamme
 * Created: March 17, 2011
 * Changed: September 20, 2011
 ********************************************************************
 * Local variables of program mnEth
 ********************************************************************)
VAR
	_xmnEthOk : BOOL;
_CfgGetBroadcastAdr : CfgGetBroadcastAddr;
END_VAR
(*Ermittlung des Ethernetinterface*)
VAR
	_GetEthPort : kgGetEthPort;
	_sEthDevice : STRING[15];
END_VAR
(*Maschinennummer*)
VAR
	_sMnr : STRING[15];
END_VAR
(*Hostname*)
VAR
	_CfgSetHostName : CfgSetHostName;
	_sHostname : STRING[15];
END_VAR
(*Defaultwerte setzen*)
VAR
	_xSetDefault : BOOL;
END_VAR
(*Werte vom USB*)
VAR
	_FileOpenCsv : FileOpen;
END_VAR
(*Parsen allgemein*)
VAR
	_sPathCsv : STRING[127];
	_MemPartCreate : AsMemPartCreate;
	_MemPartAlloc : AsMemPartAlloc;
	_pParseMem : UDINT;
	_FileReadCsv : FileRead;
	_FileCloseCsv : FileClose;
	_GetCsvDat : mnParam_GetCsvDat;
	_lFileSize : UDINT;
END_VAR
(*Hilfsvariablen*)
VAR
	_ParSet : _EthPar_typ;
	_lIPAdr : UDINT;
	_pOctet : REFERENCE TO ARRAY[0..3] OF USINT;
	_lGatewayAdr : UDINT;
	_DirInfo : DirInfo;
	_DirCreate : DirCreate;
	_lBroadcastAdr : UDINT;
	_sBroadcastAdr : STRING[15];
	_xChanged : BOOL;
END_VAR
(*Werte von CF*)
VAR
	_ParSetCF : _EthPar_typ;
	_xSetIPFromCF : BOOL;
END_VAR
(*Funktionen*)
VAR
	_CfgSetSubnetMask : CfgSetSubnetMask;
	_CfgSetIPAddr : CfgSetIPAddr;
	_CfgSetDefaultGateway : CfgSetDefaultGateway;
	_CfgSetBroadcastAdr : CfgSetBroadcastAddr;
	_CfgGetGateway : CfgGetDefaultGateway;
	_CfgGetIPAddress : CfgGetIPAddr;
END_VAR
(*Werte schreiben*)
VAR
	_WriteBOM : mnParam_WriteBOM_Mem;
	_WriteCsv90 : mnParam_WriteCSV90_Mem;
	_IPRow : mnParam_CsvIPRow_typ;
	_FileDeleteCsv : FileDelete;
	_FileCreateCsv : FileCreate;
	_FileWriteCsv : FileWrite;
END_VAR
(*Zyklisch*)
VAR
	_ParGet : _EthPar_typ;
	_ParAktuell : _EthPar_typ;
	enEState : enumEthernetState;
	_TONidle : TON;
	_TONwarning : TON;
	_bWaitCounter : USINT;
END_VAR
(*Konstanten*)
VAR CONSTANT
	_MNETH_MSG_IFDEVICE : UINT := 20000;
	_MNETH_MSG_MEM : UINT := 20001;
	_MNETH_MSG_SETDEF : UINT := 20100;
	_MNETH_MSG_WRITECSV : UINT := 20101;
	_MNETH_MSG_CHANGE : UINT := 20102;
	_MNETH_MSG_SETUSB : UINT := 20103;
END_VAR
VAR
	_lPosLF : UDINT;
	_lPosCR : UDINT;
	_kgMachineTypeW3 : kgMachinetypeW3_typ;
	_lNetId : UDINT;
	_cfgLease : cfgLease_typ;
	_CfgSetDhcpsData : CfgSetDhcpsData;
	_xDHCPstarted : BOOL;
	_CfgSetDhcpServer : CfgSetDhcpServer;
	_xSNTPSrvStarted : BOOL;
	_xSNTPCltStarted : BOOL;
	_CfgSetSntpClient : CfgSetSntpClient;
	_CfgSetSntpServer : CfgSetSntpServer;
	_sSubnetMask : STRING[15] := '255.255.240.000';
	_xSetHostname : BOOL := TRUE;
	_CfgGetHostName : CfgGetHostName;
	_sActHostname : STRING[15];
	_sActBroadcastAdr : STRING[15];
	_sActIPAdr : STRING[15];
	_sActGateway : STRING[15];
	_sPkgName : STRING[11];
	_VerStruc : MoVerStruc_typ;
	_kgMsgStatus : kgMsg_Status_Typ;
	_xCheckedUSB : BOOL := FALSE;
	_sDevice : STRING[31];
END_VAR
```

### Pkg_mnEth_History.txt
```
2.01.0	2011-09-07	AH Änderung der Standardnetzwerkmaske auf 20 bit
2.02.0	2011-09-20	AH Schaut jetzt auf mnParamStatAd.xParamOK, setzt Version 0.5 von mnParam voraus
2.02.1	2011-09-28	AH Interface für PCTs korregiert
2.03.0	2011-10-06	AH Maschinennummer aus _Info_, IP-Adresse usw. NONVOLATILE
2.04.0	2011-10-20	AH Umstellung auf AS 3.0.90
2.05.0	2012-01-10	AH PackageVersion wird nun in mnEthStatAd angezeigt
2.06.0	2012-01-27	AH Unabhängig von NetLink
2.07.0	2012-02-03	AH Es wird kein USB-Stick mehr als Device gelinkt. Es wird vorausgesetzt, dass die
					   Devices (Siehe Konstanten KG_DEVICE_USBSTICK1 und KG_DEVICE_USBSTICK2 bereits
					   in der sysconf festgelegt sind) Setzt KGStandard 1.14.0 voraus.
2.08.0	2012-02-08	AH Kompatibel zu KGStandard 1.15.0 (KGstdLib 1.03.0)
2.09.0	2012-02-23	AH Kompatibel zu hlKanLink 0.94.0
					   - Hostname auf 15 Zeichen gekürzt
					   Kompatibel mit mnTest
2.09.1	2012-03-20	AH Abhängigkeiten ergänzt
2.10.0	2012-05-11	AH Auswertung USB in den zyklischen Teil gelegt.
2.10.1	2012-07-17	AH Filehandle wurde nach Create nicht freigegeben.
```

### CfgMsgStat.mnEth.txt
```
;****************************
; System Manager
;*****************************
00004, 20000, 00000, 00000;
00004, 20001, 00000, 00000;
00004, 20100, 00000, 00000;
00004, 20101, 00000, 00000;
00004, 20102, 00000, 00000;
00004, 20103, 00000, 00000;
```

### Package Logical/Standard/Kanlink/KGFramework/Pkg_mnCnt - Management-Ebene für Zähler

### Pkg_mnCnt.typ - Global data types
```iecst
(********************************************************************
 * COPYRIGHT -- Microsoft
 ********************************************************************
 * Package: Pkg_mnCnt
 * File: Pkg_mnCnt.typ
 * Author: hunholz
 * Created: July 02, 2011
 ********************************************************************
 * Data types of package Pkg_mnCnt
 ********************************************************************)

TYPE
	mnCntLocation_Typ : 	STRUCT
		sNameId : STRING[10]; (*Text-ID des Ortes*)
		bLocationExt : USINT; (*0 - Interner Ort, 1 - Externer Ort*)
	END_STRUCT;
	mnCntStatAd_Typ : 	STRUCT
		sPkgVersion : STRING[10];
	END_STRUCT;
	mnCntEventBatch_Typ : 	STRUCT
		Batch : BatchData_typ;
		FromLocation : mnCntLocation_Typ;
		ToLocation : mnCntLocation_Typ;
		bProgram : USINT;
		bEvent : USINT; (*0 - Beladung, 1 - Entladung, 2 - Geändert, 3 - Gelöscht*)
	END_STRUCT;
	mnCntEventCounter_Typ : 	STRUCT
		Source : mnCntLocation_Typ; (*Quell Ort für Medien*)
		Destination : mnCntLocation_Typ; (*Ziel Ort für Medien, Ort der Messung*)
		BatchNo : GUID_type; (*Postennummer (long oder GUID)*)
		dtTimeStamp : DATE_AND_TIME; (*Zeitstempel des Zählwerts*)
		lAmount : UDINT; (*Menge bzw. Wert*)
		lNomAmount : UDINT; (*Sollmenge*)
		bTypeBatchNo : USINT; (*0 - Postennummer ist long, 1 - Postennummer ist GUID*)
		bType : USINT; (*1 - Wasser, 2 - Dampf, 3 - Gas, 4 - Elektrische Energie, 11 - Temperatur, 12 - Druck, 13 - Drehzahl*)
	END_STRUCT;
	mnCntEventDosing_Typ : 	STRUCT
		BatchNo : GUID_type; (*Postennummer (long oder GUID)*)
		dtTimeStamp : DATE_AND_TIME; (*Zeitstempel der Dosierung*)
		rNomAmount : REAL; (*Solldosiermenge*)
		rAmount : REAL; (*Istdosiermenge*)
		rPumpConst : REAL; (*Pumpenkonstante*)
		sUnit : STRING[11]; (*Einheit der Dosierung*)
		utfName : WSTRING[23]; (*Name der Dosierung*)
		Source : mnCntLocation_Typ; (*Quelle*)
		Destination : mnCntLocation_Typ; (*Zielort*)
		bTypeBatchNo : USINT; (*0 - Postennummer ist long, 1 - Postennummer ist GUID*)
	END_STRUCT;
	mnCntEventDosingId_Typ : 	STRUCT
		bId : USINT;
		DosingEvent : mnCntEventDosing_Typ;
	END_STRUCT;
	IFmnCnt_Typ : 	STRUCT
		In : IFmnCntIn_Typ;
		Out : IFmnCntOut_Typ;
	END_STRUCT;
	mnCntEventTime_Typ : 	STRUCT
		dtTimeStamp : DATE_AND_TIME;
		lAmount : UDINT; (*Zeitintervall*)
		bState : USINT; (*0 - Inaktiv, 1 - Warten, 2 - Aktiv*)
		bSubState : USINT; (*0.0 - AUS/Taktende, 0.1 - Stop, 0.2 - int. Störung, 0.3 - ext. Störung, 0.4 - Sicherer Halt, 0.5 - NOT-HALT, 1.0 - Beladung, 1.1 - Entladung, 1.2 - Dosierung, 2.0 - Prozess, 2.1 - Vorbereitung*)
	END_STRUCT;
	IFmnCntOut_Typ : 	STRUCT
		wStatus : UINT;
		xBatchEventReadOK : BOOL;
		xCounterEventReadOK : ARRAY[0..MNCNT_IDX_COUNTER_MAX]OF BOOL;
		xDosingEventReadOK : ARRAY[1..48]OF BOOL;
		xTimeEventReadOK : BOOL;
	END_STRUCT;
	IFmnCntIn_Typ : 	STRUCT
		wCmd : UINT;
		bBatchEventValid : USINT; (*0->1: Batchevent übernehmen*)
		bCntEventValid : ARRAY[0..MNCNT_IDX_COUNTER_MAX]OF USINT; (*0->1 : Zählerwert übernehmen*)
		bDosingEventValid : ARRAY[1..48]OF USINT; (*0->1 : Zählerwert übernehmen*)
		bTimeEventValid : USINT; (*0->1 : Zeitwert übernehmen*)
		BatchEvent : mnCntEventBatch_Typ; (*Postenevent*)
		CounterEvent : ARRAY[0..MNCNT_IDX_COUNTER_MAX]OF mnCntEventCounter_Typ; (*Zählerevents*)
		DosingEvent : ARRAY[1..48]OF mnCntEventDosing_Typ; (*max. 48 Dosierevents*)
		TimeEvent : mnCntEventTime_Typ; (*Zeitwerte*)
	END_STRUCT;
	mnCntParMacDosingDef_Typ : 	STRUCT
		utfName : WSTRING[23];
		xUseConversion : BOOL;
		bCompartment : USINT;
		bIdx : USINT;
		bReserve : USINT;
		rConversionMultiplier : REAL;
		sUnit : STRING[11];
	END_STRUCT;
	mnCntParMac_Typ : 	STRUCT
		DosingDefines : ARRAY[1..48]OF mnCntParMacDosingDef_Typ;
	END_STRUCT;
	mnCntPar_Typ : 	STRUCT
		Mac : mnCntParMac_Typ;
	END_STRUCT;
END_TYPE
```

### Pkg_mnCnt.var - Global variables
```iecst
(********************************************************************
 * COPYRIGHT -- Microsoft
 ********************************************************************
 * Package: Pkg_mnCnt
 * File: Pkg_mnCnt.var
 * Author: hunholz
 * Created: July 02, 2011
 ********************************************************************
 * Variables of package Pkg_mnCnt
 ********************************************************************)
VAR
	IFmnCnt : IFmnCnt_Typ := (0);
	mnCntCmd : KG_Cmd_typ := (0);
	mnCntPar : mnCntPar_Typ := (0);
	mnCntStatAd : mnCntStatAd_Typ;
END_VAR
(*Konstanten*)
VAR CONSTANT
	MNCNT_MSG_READ_SUM : UINT := 1000;
	MNCNT_MSG_DELETE_SUM : UINT := 1001;
	MNCNT_MSG_CREATE_SUM : UINT := 1002;
	MNCNT_MSG_INFO_SUM : UINT := 1003;
	MNCNT_MSG_CREATE_RB : UINT := 1004;
	MNCNT_MSG_INFO_RB : UINT := 1005;
	MNCNT_MSG_CFG : UINT := 1006;
	MNCNT_MSG_CNT_CFG : UINT := 1007;
	MNCNT_MSG_RB_NEW : UINT := 1009;
	MNCNT_BATCHEVENT_LOAD : USINT := 0; (*Postenevent bei Beladung*)
	MNCNT_BATCHEVENT_UNLOAD : USINT := 1; (*Postenevent bei Entladung*)
	MNCNT_BATCHEVENT_CHANGEDATA : USINT := 2; (*Postenevent bei Datenänderung*)
	MNCNT_BATCHEVENT_DELETE : USINT := 3; (*Postenevent zum Löschen eines Postens*)
	MNCNT_COUNTERTYPE_WATER : USINT := 1; (*Wasserzähler*)
	MNCNT_COUNTERTYPE_STEAM : USINT := 2; (*Dampf*)
	MNCNT_COUNTERTYPE_GAS : USINT := 3; (*Gas*)
	MNCNT_COUNTERTYPE_ELECTRICENERGY : USINT := 4; (*Elektrische Energie*)
	MNCNT_COUNTERTYPE_NOTCOUNTABLE : USINT := 11; (*Nicht zählbare Werte*)
	MNCNT_COUNTERTYPE_TEMPERATURE : USINT := 11; (*Temperatur*)
	MNCNT_COUNTERTYPE_PRESSURE : USINT := 12; (*Druck*)
	MNCNT_COUNTERTYPE_RPM : USINT := 13; (*Drehzahl*)
	MNCNT_IDX_TIMESTATE_MAX : UINT := 2; (*0 - PAUSED, 1 - WAIT, 2 - ACTIVE*)
	MNCNT_TIMERSTATE_PAUSED : USINT := 0;
	MNCNT_TIMERSTATE_WAIT : USINT := 1;
	MNCNT_TIMERSTATE_ACTIVE : USINT := 2;
	MNCNT_IDX_TIMESUBSTATE_MAX : UINT := 6;
	MNCNT_TIMERSUBSTATE_PROCESSING : USINT := 0;
	MNCNT_TIMERSUBSTATE_WASHING : USINT := 0;
	MNCNT_TIMERSUBSTATE_PREPERATION : USINT := 1;
	MNCNT_TIMERSUBSTATE_TRANSFER : USINT := 2;
	MNCNT_TIMERSUBSTATE_PREPFORSTOP : USINT := 3;
	MNCNT_TIMERSUBSTATE_LOADING : USINT := 0;
	MNCNT_TIMERSUBSTATE_UNLOADING : USINT := 1;
	MNCNT_TIMERSUBSTATE_DOSING : USINT := 2;
	MNCNT_TIMERSUBSTATE_WATERLEVEL : USINT := 3;
	MNCNT_TIMERSUBSTATE_TEMPERATURE : USINT := 4;
	MNCNT_TIMERSUBSTATE_DISINFECTION : USINT := 5;
	MNCNT_TIMERSUBSTATE_AIRPRESSURE : USINT := 6;
	MNCNT_TIMERSUBSTATE_OFF : USINT := 0;
	MNCNT_TIMERSUBSTATE_STOP : USINT := 1;
	MNCNT_TIMERSUBSTATE_INTFAULT : USINT := 2;
	MNCNT_TIMERSUBSTATE_EXTFAULT : USINT := 3;
	MNCNT_TIMERSUBSTATE_SAFESTOP : USINT := 4;
	MNCNT_TIMERSUBSTATE_EMERGENCYSTP : USINT := 5;
END_VAR
```

### Program Logical/Standard/Kanlink/KGFramework/Pkg_mnCnt/mnCnt (IEC) - Counter Manager
